(* LS Electric XG5000 project: POL(230517) *)
(* PLC NewPLC *)
(* module base 0 slot 0: FEnet:XGL-EFMT(B) (Fast Ethernet 통신 모듈, 전기 Master) *)
(* module base 1 slot 0: 아날로그입력 모듈:XGF-AC8A (A/D 전류 입력형 8채널) *)
(* module base 1 slot 1: 입력 모듈:XGI-D28A/B (DC 24V 입력, 64점 (전류소스 싱크공용/ 전류소스 입력)) *)
(* module base 1 slot 2: 입력 모듈:XGI-D28A/B (DC 24V 입력, 64점 (전류소스 싱크공용/ 전류소스 입력)) *)
(* module base 1 slot 3: 입력 모듈:XGI-D28A/B (DC 24V 입력, 64점 (전류소스 싱크공용/ 전류소스 입력)) *)
(* module base 1 slot 4: 입력 모듈:XGI-D28A/B (DC 24V 입력, 64점 (전류소스 싱크공용/ 전류소스 입력)) *)
(* module base 1 slot 5: 입력 모듈:XGI-D28A/B (DC 24V 입력, 64점 (전류소스 싱크공용/ 전류소스 입력)) *)
(* module base 1 slot 6: 출력 모듈:XGQ-TR8A/B (트랜지스터 출력, 64점 (0.1A용, 싱크출력/소스출력)) *)
(* module base 1 slot 7: 출력 모듈:XGQ-TR8A/B (트랜지스터 출력, 64점 (0.1A용, 싱크출력/소스출력)) *)
(* module base 2 slot 0: 출력 모듈:XGQ-TR8A/B (트랜지스터 출력, 64점 (0.1A용, 싱크출력/소스출력)) *)
(* module base 2 slot 1: 출력 모듈:XGQ-TR8A/B (트랜지스터 출력, 64점 (0.1A용, 싱크출력/소스출력)) *)
(* module base 2 slot 2: 출력 모듈:XGQ-TR8A/B (트랜지스터 출력, 64점 (0.1A용, 싱크출력/소스출력)) *)
(* module base 2 slot 3: 입력 모듈:XGI-D28A/B (DC 24V 입력, 64점 (전류소스 싱크공용/ 전류소스 입력)) *)
(* module base 2 slot 4: 입력 모듈:XGI-D28A/B (DC 24V 입력, 64점 (전류소스 싱크공용/ 전류소스 입력)) *)
(* module base 2 slot 5: 입력 모듈:XGI-D28A/B (DC 24V 입력, 64점 (전류소스 싱크공용/ 전류소스 입력)) *)
(* module base 2 slot 6: 출력 모듈:XGQ-TR8A/B (트랜지스터 출력, 64점 (0.1A용, 싱크출력/소스출력)) *)
(* module base 2 slot 7: Cnet:XGL-C42A/B (Cnet 통신 모듈(RS-422/485, RS-422/485)) *)
(* module base 2 slot 8: 아날로그출력 모듈:XGF-DC4A (D/A 전류 출력형 4채널) *)
VAR_GLOBAL
    TK101H : DWORD;
    TK101HH : DWORD;
    TK101L : DWORD;
    TK101LL : DWORD;
    TK101VAL : DWORD;
    TK102H : DWORD;
    TK102HH : DWORD;
    TK102L : DWORD;
    TK102LL : DWORD;
    TK102VAL : DWORD;
    TK103H : DWORD;
    TK103HH : DWORD;
    TK103L : DWORD;
    TK103LL : DWORD;
    TK103VAL : DWORD;
    TK104H : DWORD;
    TK104HH : DWORD;
    TK104L : DWORD;
    TK104LL : DWORD;
    TK104VAL : DWORD;
    TK105H : DWORD;
    TK105HH : DWORD;
    TK105L : DWORD;
    TK105LL : DWORD;
    TK105VAL : DWORD;
    TK106H : DWORD;
    TK106HH : DWORD;
    TK106L : DWORD;
    TK106LL : DWORD;
    TK106VAL : DWORD;
    TK107H : DWORD;
    TK107HH : DWORD;
    TK107L : DWORD;
    TK107LL : DWORD;
    TK107VAL : DWORD;
    TK108H : DWORD;
    TK108HH : DWORD;
    TK108L : DWORD;
    TK108LL : DWORD;
    TK108VAL : DWORD;
    TK109H : DWORD;
    TK109HH : DWORD;
    TK109L : DWORD;
    TK109LL : DWORD;
    TK109VAL : DWORD;
    TK110H : DWORD;
    TK110HH : DWORD;
    TK110L : DWORD;
    TK110LL : DWORD;
    TK110VAL : DWORD;
    TK111H : DWORD;
    TK111HH : DWORD;
    TK111L : DWORD;
    TK111LL : DWORD;
    TK111VAL : DWORD;
    TK112H : DWORD;
    TK112HH : DWORD;
    TK112L : DWORD;
    TK112LL : DWORD;
    TK112VAL : DWORD;
    TK113H : DWORD;
    TK113HH : DWORD;
    TK113L : DWORD;
    TK113LL : DWORD;
    TK113VAL : DWORD;
    _0000_ADDR_LNM AT %LW3761 : WORD; (* FEnet: LNM 정보(Ver 6.0이상) *)
    _0000_LINE_TOPOLOGY AT %LX60148 : BOOL; (* FEnet: Line topology 상태(Ver 6.0이상) *)
    _0100_CH0_ACT AT %UX1.0.16 : BOOL; (* 아날로그입력 모듈: 채널0 운전중 *)
    _0100_CH0_DATA AT %UW1.0.2 : INT; (* 아날로그입력 모듈: 채널0 변환값 *)
    _0100_CH0_IDD AT %UX1.0.160 : BOOL; (* 아날로그입력 모듈: 채널0 입력단선검출 *)
    _0100_CH1_ACT AT %UX1.0.17 : BOOL; (* 아날로그입력 모듈: 채널1 운전중 *)
    _0100_CH1_DATA AT %UW1.0.3 : INT; (* 아날로그입력 모듈: 채널1 변환값 *)
    _0100_CH1_IDD AT %UX1.0.161 : BOOL; (* 아날로그입력 모듈: 채널1 입력단선검출 *)
    _0100_CH2_ACT AT %UX1.0.18 : BOOL; (* 아날로그입력 모듈: 채널2 운전중 *)
    _0100_CH2_DATA AT %UW1.0.4 : INT; (* 아날로그입력 모듈: 채널2 변환값 *)
    _0100_CH2_IDD AT %UX1.0.162 : BOOL; (* 아날로그입력 모듈: 채널2 입력단선검출 *)
    _0100_CH3_ACT AT %UX1.0.19 : BOOL; (* 아날로그입력 모듈: 채널3 운전중 *)
    _0100_CH3_DATA AT %UW1.0.5 : INT; (* 아날로그입력 모듈: 채널3 변환값 *)
    _0100_CH3_IDD AT %UX1.0.163 : BOOL; (* 아날로그입력 모듈: 채널3 입력단선검출 *)
    _0100_CH4_ACT AT %UX1.0.20 : BOOL; (* 아날로그입력 모듈: 채널4 운전중 *)
    _0100_CH4_DATA AT %UW1.0.6 : INT; (* 아날로그입력 모듈: 채널4 변환값 *)
    _0100_CH4_IDD AT %UX1.0.164 : BOOL; (* 아날로그입력 모듈: 채널4 입력단선검출 *)
    _0100_CH5_ACT AT %UX1.0.21 : BOOL; (* 아날로그입력 모듈: 채널5 운전중 *)
    _0100_CH5_DATA AT %UW1.0.7 : INT; (* 아날로그입력 모듈: 채널5 변환값 *)
    _0100_CH5_IDD AT %UX1.0.165 : BOOL; (* 아날로그입력 모듈: 채널5 입력단선검출 *)
    _0100_CH6_ACT AT %UX1.0.22 : BOOL; (* 아날로그입력 모듈: 채널6 운전중 *)
    _0100_CH6_DATA AT %UW1.0.8 : INT; (* 아날로그입력 모듈: 채널6 변환값 *)
    _0100_CH6_IDD AT %UX1.0.166 : BOOL; (* 아날로그입력 모듈: 채널6 입력단선검출 *)
    _0100_CH7_ACT AT %UX1.0.23 : BOOL; (* 아날로그입력 모듈: 채널7 운전중 *)
    _0100_CH7_DATA AT %UW1.0.9 : INT; (* 아날로그입력 모듈: 채널7 변환값 *)
    _0100_CH7_IDD AT %UX1.0.167 : BOOL; (* 아날로그입력 모듈: 채널7 입력단선검출 *)
    _0208_CH0_ACT AT %UX2.8.16 : BOOL; (* 아날로그출력 모듈: 채널0 운전중 *)
    _0208_CH0_DATA AT %UW2.8.3 : INT; (* 아날로그출력 모듈: 채널0 입력값 *)
    _0208_CH0_ERR AT %UX2.8.0 : BOOL; (* 아날로그출력 모듈: 채널0 에러 *)
    _0208_CH0_OUTEN AT %UX2.8.32 : BOOL; (* 아날로그출력 모듈: 채널0 출력상태설정 *)
    _Auto_re_count : BOOL;
END_VAR

(* Comments on direct variables
%IX1.1.0	Power 0n_PB
%IX1.1.1	Power Off_PB
%IX1.1.2	Scada 선택 SL
%IX1.1.3	Panel 선택 SL
%IX1.1.5	Manual On_PB
%IX1.1.6	Auto On_PB
%IX1.1.7	Lamp Test PB
%IX1.1.8	Auto Stop (PANEL)
%IX1.1.9	Horn Reset PB
%IX1.1.10	In-TLV21601
%IX1.1.11	In-TLV21602
%IX1.1.12	In-TLV21701
%IX1.1.13	In-TLV21702
%IX1.1.14	In-TLV21801
%IX1.1.15	BCVF Open
%IX1.1.17	EM-Stop RESET
(PANEL)
%IX1.1.18	TK1-EM
%IX1.1.19	TK2-EM
%IX1.1.20	TK3-EM
%IX1.1.21	TK4-EM
%IX1.1.22	TK5-EM
%IX1.1.23	TK6-EM
%IX1.1.24	TK7-EM
%IX1.1.25	TK8-EM
%IX1.1.26	TK9-EM
%IX1.1.27	TK10-EM
%IX1.1.28	PUMP실-EM
%IX1.1.31	MAIN PANEL-EM PB
%IX1.1.32	TK-101 HLV  선택 PB
%IX1.1.33	VENT1 Trouble 
%IX1.1.34	VENT1 TURN 
%IX1.1.35	P101A OCR
%IX1.1.36	P101A Local Ready
%IX1.1.37	P101A Stop PB
%IX1.1.38	P101A Run PB
%IX1.1.39	P101B OCR
%IX1.1.40	P101B Local Ready
%IX1.1.41	P101B Stop_PB
%IX1.1.42	P101B Run_PB
%IX1.1.43	P101C OCR
%IX1.1.44	P101C Local Ready
%IX1.1.45	P101C Stop_PB
%IX1.1.46	P101C Run_PB
%IX1.1.47	TK-101 Clearance
%IX1.1.48	TK-102 HLV  선택 PB
%IX1.1.49	Vent2 Trouble
%IX1.1.50	Vent2 On
%IX1.1.51	P102A OCR
%IX1.1.52	P102A Local Ready
%IX1.1.53	P102A Stop_PB
%IX1.1.54	P102A Run_PB
%IX1.1.55	P102B OCR
%IX1.1.56	P102B Local Ready
%IX1.1.57	P102B Stop_PB
%IX1.1.58	P102B Run_PB
%IX1.1.59	P102C OCR
%IX1.1.60	P102C Local Ready
%IX1.1.61	P102C Stop_PB
%IX1.1.62	P102C Run_PB
%IX1.1.63	TK-102 Clearance
%IX1.2.0	TK-103 HLV 선택 PB
%IX1.2.1	Vent3 Trouble_in
%IX1.2.2	Vent3 On_in
%IX1.2.3	P103A OCR
%IX1.2.4	P103A Local Ready
%IX1.2.5	P103A Stop_PB
%IX1.2.6	P103A Run_PB
%IX1.2.7	P103B OCR
%IX1.2.8	P103B Local Ready
%IX1.2.9	P103B Stop_PB
%IX1.2.10	P103B Run_PB
%IX1.2.11	P103C OCR
%IX1.2.12	P103C Local Ready
%IX1.2.13	P103C Stop_PB
%IX1.2.14	P103C Run_PB
%IX1.2.15	TK-103 Clearance
%IX1.2.16	TK-104 HLV 선택 PB
%IX1.2.17	Vent4 Trouble_in
%IX1.2.18	Vent4 On_in
%IX1.2.19	P104A OCR
%IX1.2.20	P104A Local Ready
%IX1.2.21	P104A Stop_PB
%IX1.2.22	P104A Run_PB
%IX1.2.23	P104B OCR
%IX1.2.24	P104B Local Ready
%IX1.2.25	P104B Stop_PB
%IX1.2.26	P104B Run_PB
%IX1.2.27	P104C OCR
%IX1.2.28	P104C Local Ready
%IX1.2.29	P104C Stop_PB
%IX1.2.30	P104C Run_PB
%IX1.2.31	TK-104 Clearance
%IX1.2.32	TK-105 선택 [Panel]
%IX1.2.33	Vent5 Trouble_in
%IX1.2.34	Vent5 On_in
%IX1.2.35	P105A OCR
%IX1.2.36	P105A Local Ready
%IX1.2.37	P105A Stop_PB
%IX1.2.38	P105A Run_PB
%IX1.2.39	P105B OCR
%IX1.2.40	P105B Local Ready
%IX1.2.41	P105B Stop_PB
%IX1.2.42	P105B Run_PB
%IX1.2.43	P105C OCR
%IX1.2.44	P105C Local Ready
%IX1.2.45	P105C Stop_PB
%IX1.2.46	P105C Run_PB
%IX1.2.47	TK-105 Clearance
%IX1.2.48	TK-106 선택 [Panel]
%IX1.2.49	Vent6 Trouble_in
%IX1.2.50	Vent6 On_in
%IX1.2.51	P106A OCR
%IX1.2.52	P106A Local Ready
%IX1.2.53	P106A Stop_PB
%IX1.2.54	P106A Run_PB
%IX1.2.55	P106B OCR
%IX1.2.56	P106B Local Ready
%IX1.2.57	P106B Stop_PB
%IX1.2.58	P106B Run_PB
%IX1.2.59	P106C OCR
%IX1.2.60	P106C Local Ready
%IX1.2.61	P106C Stop_PB
%IX1.2.62	P106C Run_PB
%IX1.2.63	TK-106 Clearance
%IX1.3.0	TK-107 HLV 선택PB
%IX1.3.1	Vent7 Trouble
%IX1.3.2	Vent7 On
%IX1.3.3	P107A_OCR
%IX1.3.4	P107A_Local Ready
%IX1.3.5	P107A Stop_PB
%IX1.3.6	P107A Run_PB
%IX1.3.7	P107B_OCR
%IX1.3.8	P107B Local Ready
%IX1.3.9	P107B Stop_PB
%IX1.3.10	P107B Run_PB
%IX1.3.11	P107C_OCR
%IX1.3.12	P107C Local Ready
%IX1.3.13	P107C Stop_PB
%IX1.3.14	P107C Run_PB
%IX1.3.15	TK-107 Clearance
%IX1.3.16	TK-108 HLV 선택PB
%IX1.3.17	Vent8 Trouble_in
%IX1.3.18	Vent8 On_in
%IX1.3.19	P108A_OCR
%IX1.3.20	P108A_Local Ready
%IX1.3.21	P108A Stop_PB
%IX1.3.22	P108A Run_PB
%IX1.3.23	P108B_OCR
%IX1.3.24	P108B Local Ready
%IX1.3.25	P108B Stop_PB
%IX1.3.26	P108B Run_PB
%IX1.3.27	P108C_OCR
%IX1.3.28	P108C Local Ready
%IX1.3.29	P108C Stop_PB
%IX1.3.30	P108C Run_PB
%IX1.3.31	TK-108 Clearance
%IX1.3.32	TK-109 선택 [Panel]
%IX1.3.33	Vent9 Trouble_in
%IX1.3.34	Vent9 On_in
%IX1.3.35	P109A OCR
%IX1.3.36	P109A Local Ready
%IX1.3.37	P109A Stop_PB
%IX1.3.38	P109A Run_PB
%IX1.3.39	P109B OCR
%IX1.3.40	P109B Local Ready
%IX1.3.41	P109B Stop_PB
%IX1.3.42	P109B Run_PB
%IX1.3.43	P109C OCR
%IX1.3.44	P109C Local Ready
%IX1.3.45	P109C Stop_PB
%IX1.3.46	P109C Run_PB
%IX1.3.47	TK-109 Clearance
%IX1.3.48	TK-110 선택 [Panel]
%IX1.3.49	Vent10 Trouble_in
%IX1.3.50	Vent10 On_in
%IX1.3.51	P110A OCR
%IX1.3.52	P110A Local Ready
%IX1.3.53	P110A Stop_PB
%IX1.3.54	P110A Run_PB
%IX1.3.55	P110B OCR
%IX1.3.56	P110B Local Ready
%IX1.3.57	P110B Stop_PB
%IX1.3.58	P110B Run_PB
%IX1.3.59	P110C OCR
%IX1.3.60	P110C Local Ready
%IX1.3.61	P110C Stop_PB
%IX1.3.62	P110C Run_PB
%IX1.3.63	TK-110 Clearance
%IX1.4.0	HLVD-21301 FULL
%IX1.4.1	Water21301_in
%IX1.4.2	P111 OCR
%IX1.4.3	P111 Local S/W ON
%IX1.4.4	P111 Stop_PB
%IX1.4.5	P111 Run_PB
%IX1.4.6	Drain-111
Clearance
%IX1.4.7	HLVD-21401 FULL
%IX1.4.8	Water21401_in
%IX1.4.9	P112OCR
%IX1.4.10	P112 Local Ready
%IX1.4.11	P112 Stop_PB
%IX1.4.12	P112 Run_PB
%IX1.4.13	Drain-112
Clearance
%IX1.4.14	HLVD-21501 FULL
%IX1.4.15	Water21501_in
%IX1.4.16	P113 OCR
%IX1.4.17	P113 Local Ready
%IX1.4.18	Drain-113
Clearance
%IX1.4.19	UP201A OCR
%IX1.4.20	UP201A  Local Ready
%IX1.4.21	UP201A Stop_PB
%IX1.4.22	UP201A Run_PB
(PANEL)
%IX1.4.23	UP201B OCR
%IX1.4.24	UP201B Local Ready
%IX1.4.25	UP201B Stop_PB
%IX1.4.26	UP201B Run_PB
%IX1.4.27	UP202A OCR
%IX1.4.28	UP202A Local Ready
%IX1.4.29	UP202A Stop_PB
(PANEL)
%IX1.4.30	UP202A Run_PB
(PANEL)
%IX1.4.31	UP202B OCR
%IX1.4.32	UP202B Local Ready
%IX1.4.33	UP202B Stop_PB
%IX1.4.34	UP202B Run_PB
%IX1.4.35	UP203A OCR
%IX1.4.36	UP203A Local Ready
%IX1.4.37	UP203A Stop_PB
(PANEL)
%IX1.4.38	UP203A Run_PB
(PANEL)
%IX1.4.39	UP203B OCR
%IX1.4.40	UP203B Local Ready
%IX1.4.41	UP203B Stop_PB
%IX1.4.42	UP203B Run_PB
%IX1.4.45	PIPE LINE MOV20105 Close-PB
%IX1.4.47	PIPE LINE MOV 20105 Open-PB
%IX1.4.49	MOV20102 Over Torque
%IX1.4.50	MOV20102 Local
%IX1.4.51	MOV20102 Close-PB
%IX1.4.52	MOV20102 Close position
%IX1.4.53	MOV20102 Open-PB
%IX1.4.54	MOV20102 Open position
%IX1.4.55	MOV20103  Over Torque
%IX1.4.56	MOV20103  Local
%IX1.4.57	MOV20103 Close-PB
%IX1.4.58	MOV20103 Close position
%IX1.4.59	MOV20103 Open-PB
%IX1.4.60	MOV20103 Open position
%IX1.4.61	MOV20104 Over Torque
%IX1.4.62	MOV20104 Local
%IX1.4.63	MOV20104 Close-PB
%IX1.5.0	MOV20104 Close position
%IX1.5.1	MOV20104 Open-PB
%IX1.5.2	MOV20104 Open position
%IX1.5.3	MOV20105 Over Torque
%IX1.5.4	MOV20105 Local
%IX1.5.5	MOV20105 Close-PB
%IX1.5.6	MOV20105 Close position
%IX1.5.7	MOV20105 Open-PB
%IX1.5.8	MOV20105 Open position
%IX1.5.9	P101A Auto 1차 운전 선택 Switch(PANEL)
%IX1.5.10	P101B Auto 1차 운전 선택 Switch(PANEL)
%IX1.5.11	P102A Auto 1차 운전 선택 Switch(PANEL)
%IX1.5.12	P102B Auto 1차 운전 선택 Switch(PANEL)
%IX1.5.13	P103A Auto 1차 운전 선택 Switch(PANEL)
%IX1.5.14	P103B Auto 1차 운전 선택 Switch(PANEL)
%IX1.5.15	P104A Auto 1차 운전 선택 Switch(PANEL)
%IX1.5.16	P104B Auto 1차 운전 선택 Switch(PANEL)
%IX1.5.17	P107A Auto 1차 운전 선택 Switch(PANEL)
%IX1.5.18	P107B Auto 1차 운전 선택 Switch(PANEL)
%IX1.5.19	P108A Auto 1차 운전 선택 Switch(PANEL)
%IX1.5.20	P108B Auto 1차 운전 선택 Switch(PANEL)
%IX1.5.25	P101A Auto 2차 운전 선택 Switch(PANEL)
%IX1.5.26	P101B Auto 2차 운전 선택 Switch(PANEL)
%IX1.5.27	P102A Auto 2차 운전 선택 Switch(PANEL)
%IX1.5.28	P102B Auto 2차 운전 선택 Switch(PANEL)
%IX1.5.29	P103A Auto 2차 운전 선택 Switch(PANEL)
%IX1.5.30	P103B Auto 2차 운전 선택 Switch(PANEL)
%IX1.5.31	P104A Auto 2차 운전 선택 Switch(PANEL)
%IX1.5.32	P104B Auto 2차 운전 선택 Switch(PANEL)
%IX1.5.33	P107A Auto 2차 운전 선택 Switch(PANEL)
%IX1.5.34	P107B Auto 2차 운전 선택 Switch(PANEL)
%IX1.5.35	P108A Auto 2차 운전 선택 Switch(PANEL)
%IX1.5.36	P108B Auto 2차 운전 선택 Switch(PANEL)
%IX1.5.41	P113 Stop_PB
%IX1.5.42	P113 Run_PB
%IX1.5.43	Auto Start PB
%IX1.5.48	RTU#1 
OPEN SIG
TO HS_PLC
%IX1.5.49	RTU#2
OPEN SIG
TO HS_PLC
%IX1.5.50	RTU#3
OPEN SIG
TO HS_PLC
%IX1.5.51	RTU#4
OPEN SIG
TO HS_PLC
%IX1.5.52	RTU#5
OPEN SIG
TO HS_PLC
%IX1.5.53	PRV OPEN SIG TO HS_PLC
%IX2.3.0	P101A Flow Switch
%IX2.3.1	P101A THERMOSTAT
%IX2.3.2	P101B Flow Switch
%IX2.3.3	P101B THERMOSTAT
%IX2.3.4	P101C Flow Switch
%IX2.3.5	P101C Thermostat
%IX2.3.6	P102A Flow Switch
%IX2.3.7	P102A Thermostat
%IX2.3.8	P102B Flow Switch
%IX2.3.9	P102B Thermostat
%IX2.3.10	P102C Flow Switch
%IX2.3.11	P102C Thermostat
%IX2.3.12	P103A Flow Switch
%IX2.3.13	P103A Thermostat
%IX2.3.14	P103B Flow Switch
%IX2.3.15	P103B Thermostat
%IX2.3.16	P103C Flow Switch
%IX2.3.17	P103C Thermostat
%IX2.3.18	P104A Flow Switch
%IX2.3.19	P104A Thermostat
%IX2.3.20	P104B Flow Switch
%IX2.3.21	P104B Thermostat
%IX2.3.22	P104C Flow Switch
%IX2.3.23	P104C Thermostat
%IX2.3.24	UP201A Flow Switch
%IX2.3.25	UP201A Thermostat
%IX2.3.26	UP201B Flow Switch
%IX2.3.27	UP201B Thermostat
%IX2.3.28	P105A Flow Switch
%IX2.3.29	P105A Thermostat
%IX2.3.30	P105B Flow Switch
%IX2.3.31	P105B Thermostat
%IX2.3.32	P105C Flow Switch
%IX2.3.33	P105C Thermostat
%IX2.3.34	P106A Flow Switch
%IX2.3.35	P106A Thermostat
%IX2.3.36	P106B Flow Switch
%IX2.3.37	P106B Thermostat
%IX2.3.38	P106C Flow Switch
%IX2.3.39	P106C Thermostat
%IX2.3.40	P107A Flow Switch Alarm
%IX2.3.41	P107A Thermostat
%IX2.3.42	P107B Flow Switch Alarm
%IX2.3.43	P107B Thermostat
%IX2.3.44	P107C Flow Switch Alarm
%IX2.3.45	P107C Thermostat
%IX2.3.46	P108A Flow Switch Alarm
%IX2.3.47	P108A Thermostat
%IX2.3.48	P108B Flow Switch Alarm
%IX2.3.49	P108B Thermostat
%IX2.3.50	P108C Flow Switch Alarm
%IX2.3.51	P108C Thermostat
%IX2.3.52	P109A Flow Switch
%IX2.3.53	P109A Thermostat
%IX2.3.54	P109B Flow Switch
%IX2.3.55	P109B Thermostat
%IX2.3.56	P109C Flow Switch
%IX2.3.57	P109C Thermostat
%IX2.3.58	P110A Flow Switch
%IX2.3.59	P110A Thermostat
%IX2.3.60	P110B Flow Switch
%IX2.3.61	P110B Thermostat
%IX2.3.62	P110C Flow Switch
%IX2.3.63	P110C Thermostat
%IX2.4.0	P111 Flow Switch
%IX2.4.1	TK-111 Thermostat
%IX2.4.2	P112 Flow Switch
%IX2.4.3	TK-112 Thermostat
%IX2.4.4	P113 Flow Switch
%IX2.4.5	TK-113 Thermostat
%IX2.4.6	UP202A Flow Switch
%IX2.4.7	UP202A Thermostat
%IX2.4.8	UP202B Flow Switch
%IX2.4.9	UP202B Thermostat
%IX2.4.10	UP203A Flow Switch
%IX2.4.11	UP203A Thermostat
%IX2.4.12	UP203B Flow Switch
%IX2.4.13	UP203B Thermostat
%IX2.4.14	TK-101A PUMP ON MCC MC ON SIG
%IX2.4.15	TK-101B PUMP ON MCC MC ON SIG
%IX2.4.16	TK-101C PUMP ON MCC MC ON SIG
%IX2.4.17	TK-102A PUMP ON MCC MC ON SIG
%IX2.4.18	TK-102B PUMP ON MCC MC ON SIG
%IX2.4.19	TK-102C PUMP ON MCC MC ON SIG
%IX2.4.20	TK-103A PUMP ON MCC MC ON SIG
%IX2.4.21	TK-103B PUMP ON MCC MC ON SIG
%IX2.4.22	TK-103C PUMP ON MCC MC ON SIG
%IX2.4.23	TK-104A PUMP ON MCC MC ON SIG
%IX2.4.24	TK-104B PUMP ON MCC MC ON SIG
%IX2.4.25	TK-104C PUMP ON MCC MC ON SIG
%IX2.4.26	TK-105A PUMP ON MCC MC ON SIG
%IX2.4.27	TK-105B PUMP ON MCC MC ON SIG
%IX2.4.28	TK-105C PUMP ON MCC MC ON SIG
%IX2.4.29	TK-106A PUMP ON MCC MC ON SIG
%IX2.4.30	TK-106B PUMP ON MCC MC ON SIG
%IX2.4.31	TK-106C PUMP ON MCC MC ON SIG
%IX2.4.32	TK-107A PUMP ON MCC MC ON SIG
%IX2.4.33	TK-107B PUMP ON MCC MC ON SIG
%IX2.4.34	TK-107C PUMP ON MCC MC ON SIG
%IX2.4.35	TK-108A PUMP ON MCC MC ON SIG
%IX2.4.36	TK-108B PUMP ON MCC MC ON SIG
%IX2.4.37	TK-108C PUMP ON MCC MC ON SIG
%IX2.4.38	TK-109A PUMP ON MCC MC ON SIG
%IX2.4.39	TK-109B PUMP ON MCC MC ON SIG
%IX2.4.40	TK-109C PUMP ON MCC MC ON SIG
%IX2.4.41	TK-110A PUMP ON MCC MC ON SIG
%IX2.4.42	TK-110B PUMP ON MCC MC ON SIG
%IX2.4.43	TK-110C PUMP ON MCC MC ON SIG
%IX2.4.44	DRAIN TK-111 PUMP ON MCC MC ON SIG
%IX2.4.45	DRAIN TK-112 PUMP ON MCC MC ON SIG
%IX2.4.46	DRAIN TK-113 PUMP ON MCC MC ON SIG
%IX2.4.47	UP201A PUMP ON MCC MC ON SIG
%IX2.4.48	UP201B PUMP ON MCC MC ON SIG
%IX2.4.49	UP202A PUMP ON MCC MC ON SIG
%IX2.4.50	UP202B PUMP ON MCC MC ON SIG
%IX2.4.51	UP203A PUMP ON MCC MC ON SIG
%IX2.4.52	UP203B PUMP ON MCC MC ON SIG
%IX2.4.53	UP201A  Local Ready   (PANTO_1)
%IX2.4.54	UP201A RUN_PB
(PANTO_1)
%IX2.4.55	UP201A STOP_PB
(PANTO_1)
%IX2.4.56	PANTO1_EM
%IX2.4.57	UP201B  Local Ready   (PANTO_2)
%IX2.4.58	UP201B RUN_PB
(PANTO_2)
%IX2.4.59	UP201B STOP_PB
(PANTO_2)
%IX2.4.60	PANTO2_EM
%IX2.4.61	UP202A  Local Ready   (PANTO_3)
%IX2.4.62	UP202A RUN_PB
(PANTO_3)
%IX2.4.63	UP202A STOP_PB
(PANTO_3)
%IX2.5.0	PANTO3_EM
%IX2.5.1	UP203A  Local Ready   (PANTO_4)
%IX2.5.2	UP203A RUN_PB
(PANTO_4)
%IX2.5.3	UP203A STOP_PB
(PANTO_4)
%IX2.5.4	PANTO4_EM
%IX2.5.5	UP203B  Local Ready   (PANTO_5)
%IX2.5.6	UP203B RUN_PB
(PANTO_5)
%IX2.5.7	UP203B STOP_PB
(PANTO_5)
%IX2.5.8	PANTO5_EM
%IX2.5.9	Drain TK-111 Pressure SW
%IX2.5.10	Drain TK-112 Pressure SW
%IX2.5.11	Drain TK-113 Pressure SW
%IX2.5.12	LDS ALARM
%IX2.5.13	LDS PNL EM
%IX2.5.14	TK-108 LEAK - 1 ON
%IX2.5.15	TK-108 LEAK - 2 ON
%IX2.5.16	TK-108 LEAK - 3 ON
%IX2.5.17	TK-108 LEAK - 4 ON
%QX1.6.0	Power On Lamp
%QX1.6.1	Power Off Lamp
%QX1.6.2	SCADA 선택 Lamp
%QX1.6.3	Panel 선택 Lamp
%QX1.6.4	BUZZER Stop Lamp
%QX1.6.5	Manual 선택 Lamp
%QX1.6.6	Auto 선택 Lamp
%QX1.6.7	Auto Stop Lamp
%QX1.6.8	외부 HORN
%QX1.6.9	BPCV
%QX1.6.10	CVP
%QX1.6.11	EV_SOL
%QX1.6.12	CVP Lamp
%QX1.6.13	EV Lamp
%QX1.6.14	In-TLV21601 Lamp
%QX1.6.15	In-TLV21602 Lamp
%QX1.6.16	In-TLV21701 Lamp
%QX1.6.17	In-TLV21702 Lamp
%QX1.6.18	In-TLV21801Lamp
%QX1.6.19	BCVF 20101 Lamp
%QX1.6.20	BPCV Lamp
%QX1.6.21	TK103-EM Lamp
%QX1.6.22	TK104-EM Lamp
%QX1.6.23	TK105-EM Lamp
%QX1.6.24	TK106-EM Lamp
%QX1.6.25	TK107-EM Lamp
%QX1.6.26	TK108-EM Lamp
%QX1.6.27	TK109-EM Lamp
%QX1.6.28	TK110-EM Lamp
%QX1.6.29	TK101-EM Lamp
%QX1.6.30	TK102-EM Lamp
%QX1.6.31	EM-Stop RESET Lamp
%QX1.6.32	MAIN PANEL EM Lamp
%QX1.6.33	Lamp Test Lamp
%QX1.6.34	Auto Start Lamp
%QX1.6.38	PIT_01A
TROUBLE
[회수압력]
%QX1.6.39	PIT_01B
TROUBLE
[수령압력]
%QX1.6.40	PIT_02A
TROUBLE
[불출압력]
%QX1.6.41	PIT_02B
TROUBLE
[불출압력]
%QX1.6.42	FIT_01A
TROUBLE
[불출유량]
%QX1.6.43	FIT_01B
TROUBLE
[불출유량]
%QX1.6.44	FIT_03A
TROUBLE
[회수유량]
%QX1.6.45	FIT_03B
TROUBLE
[회수유량]
%QX1.6.46	A-SIDE PLC RUN Lamp
%QX1.6.47	B-SIDE PLC RUN Lamp
%QX1.6.48	HLV20301 TK101 Open
%QX1.6.49	VENT1 Trouble Lamp
%QX1.6.50	VENT1 TURN Lamp
%QX1.6.51	P101A Trouble Lamp
%QX1.6.52	P101A Local Lamp
%QX1.6.53	P101A Stop Lamp
%QX1.6.54	P101A Run
%QX1.6.55	P101B Trouble Lamp
%QX1.6.56	P101B Local Lamp
%QX1.6.57	P101B Stop Lamp
%QX1.6.58	P101B Run
%QX1.6.59	P101C Trouble Lamp
%QX1.6.60	P101C Local Lamp
%QX1.6.61	P101C Stop Lamp
%QX1.6.62	P101C Run
%QX1.6.63	HLV20401 TK102 Open
%QX1.7.0	Vent2 Trouble Lamp
%QX1.7.1	TK102 Ventilator Lamp
%QX1.7.2	P102A Trouble Lamp
%QX1.7.3	P102A Local Lamp
%QX1.7.4	P102A Stop Lamp
%QX1.7.5	P102A Run
%QX1.7.6	P102B Trouble Lamp
%QX1.7.7	P102B Local Lamp
%QX1.7.8	P102B Stop Lamp
%QX1.7.9	P102B Run
%QX1.7.10	P102C Trouble Lamp
%QX1.7.11	P102C Local Lamp
%QX1.7.12	P102C Stop Lamp
%QX1.7.13	P102C Run
%QX1.7.14	HLV20501 TK103 Open
%QX1.7.15	Vent3 Trouble Lamp
%QX1.7.16	TK103 Ventilator Lamp
%QX1.7.17	P103A Trouble Lamp
%QX1.7.18	P103A Local Lamp
%QX1.7.19	P103A Stop Lamp
%QX1.7.20	P103A Run
%QX1.7.21	P103B Trouble Lamp
%QX1.7.22	P103B Local Lamp
%QX1.7.23	P103B Stop Lamp
%QX1.7.24	P103B Run
%QX1.7.25	P103C Trouble Lamp
%QX1.7.26	P103C Local Lamp
%QX1.7.27	P103C Stop Lamp
%QX1.7.28	P103C Run
%QX1.7.29	HLV20601 TK104 Open
%QX1.7.30	Vent4 Trouble Lamp
%QX1.7.31	TK104 Ventilator Lamp
%QX1.7.32	P104A Trouble Lamp
%QX1.7.33	P104A Local Lamp
%QX1.7.34	P104A Stop Lamp
%QX1.7.35	P104A Run
%QX1.7.36	P104B Trouble Lamp
%QX1.7.37	P104B Local Lamp
%QX1.7.38	P104B Stop Lamp
%QX1.7.39	P104B Run
%QX1.7.40	P104C Trouble Lamp
%QX1.7.41	P104C Local Lamp
%QX1.7.42	P104C Stop Lamp
%QX1.7.43	P104C Run
%QX1.7.44	HLV20701 TK105 Open
%QX1.7.45	Vent5 Trouble Lamp
%QX1.7.46	TK105 Ventilator Lamp
%QX1.7.47	P105A Trouble Lamp
%QX1.7.48	P105A Local Lamp
%QX1.7.49	P105A Stop Lamp
%QX1.7.50	P105A Run 
%QX1.7.51	P105B Trouble Lamp
%QX1.7.52	P105B Local Lamp
%QX1.7.53	P105B Stop Lamp
%QX1.7.54	P105B Run
%QX1.7.55	P105C Trouble Lamp
%QX1.7.56	P105C Local Lamp
%QX1.7.57	P105C Stop Lamp
%QX1.7.58	P105C Run
%QX1.7.59	HLV20801 TK106 Open
%QX1.7.60	Vent6 Trouble Lamp
%QX1.7.61	TK106 Ventilator Lamp
%QX1.7.62	P106A Trouble Lamp
%QX1.7.63	P106A Local Lamp
%QX1.9.60	PIPE LINE MOV 20101 Trouble
%QX1.9.61	PIPE LINE MOV 20101 Local
%QX1.9.62	PIPE LINE MOV 20105 Close Lamp
%QX1.9.63	MOV20101 Close
%QX1.10.0	PIPE LINE MOV 20101 Open Lamp
%QX1.10.1	MOV20101 Open
%QX2.0.0	P106A Stop Lamp
%QX2.0.1	P106A Run
%QX2.0.2	P106B Trouble Lamp
%QX2.0.3	P106B Local Lamp
%QX2.0.4	P106B Stop Lamp
%QX2.0.5	P106B Run
%QX2.0.6	P106C Trouble Lamp
%QX2.0.7	P106C Local Lamp
%QX2.0.8	P106C Stop Lamp
%QX2.0.9	P106C Run
%QX2.0.10	HLV20901 TK107 Open
%QX2.0.11	Vent7 Trouble Lamp
%QX2.0.12	TK107 Ventilator Lamp
%QX2.0.13	P107A Trouble Lamp
%QX2.0.14	P107A Local Lamp
%QX2.0.15	P107A Stop
%QX2.0.16	P107A Run
%QX2.0.17	P107B Trouble Lamp
%QX2.0.18	P107B Local Lamp
%QX2.0.19	P107B Stop
%QX2.0.20	P107B Run
%QX2.0.21	P107C Trouble Lamp
%QX2.0.22	P107C Local Lamp
%QX2.0.23	P107C Stop
%QX2.0.24	P107C Run
%QX2.0.25	HLV21001 TK108 Open
%QX2.0.26	Vent8 Trouble Lamp
%QX2.0.27	TK108 Ventilator Lamp
%QX2.0.28	P108A Trouble Lamp
%QX2.0.29	P108A Local Lamp
%QX2.0.30	P108A Stop Lamp
%QX2.0.31	P108A Run
%QX2.0.32	P108B Trouble Lamp
%QX2.0.33	P108B Local Lamp
%QX2.0.34	P108B Stop Lamp
%QX2.0.35	P108B Run
%QX2.0.36	P108C Trouble Lamp
%QX2.0.37	P108C Local Lamp
%QX2.0.38	P108C Stop Lamp
%QX2.0.39	P108C Run
%QX2.0.40	HLV21101 TK109 Open
%QX2.0.41	Vent9 Trouble Lamp
%QX2.0.42	TK109 Ventilator
%QX2.0.43	P109A Trouble Lamp
%QX2.0.44	P109A Local Lamp
%QX2.0.45	P109A Stop Lamp
%QX2.0.46	P109A Run
%QX2.0.47	P109B Trouble Lamp
%QX2.0.48	P109B Local Lamp
%QX2.0.49	P109B Stop Lamp
%QX2.0.50	P109B Run
%QX2.0.51	P109C Trouble Lamp
%QX2.0.52	P109C Local Lamp
%QX2.0.53	P109C Stop Lamp
%QX2.0.54	P109C Run
%QX2.0.55	HLV21201 TK110 Open
%QX2.0.56	Vent10 Trouble Lamp
%QX2.0.57	TK110 Ventilator Lamp
%QX2.0.58	P110A Trouble Lamp
%QX2.0.59	P110A Local Lamp
%QX2.0.60	P110A Stop Lamp
%QX2.0.61	P110A Run
%QX2.0.62	P110B Trouble Lamp
%QX2.0.63	P110B Local Lamp
%QX2.1.0	P110B Stop Lamp
%QX2.1.1	P110B Run
%QX2.1.2	P110C Trouble Lamp
%QX2.1.3	P110C Local Lamp
%QX2.1.4	P110C Stop Lamp
%QX2.1.5	P110C Run
%QX2.1.6	HLVD FULL 21301 Lamp
%QX2.1.7	Water21301 Lamp
%QX2.1.8	P111 Trouble Lamp
%QX2.1.9	DRAIN TK-111 Local Lamp
%QX2.1.10	P111 Stop Lamp
%QX2.1.11	P111 Run
%QX2.1.12	DRAIN TANK111 Level 95%   HH Lamp
%QX2.1.13	DRAIN TANK111 Level 90%   H Lamp
%QX2.1.14	DRAIN TANK111 Level 정상 Lamp
%QX2.1.15	DRAIN TANK111 Level 15%   L  Lamp
%QX2.1.16	DRAIN TANK111 Level 10%   LL Lamp
%QX2.1.17	HLVD MAX 21401 Lamp
%QX2.1.18	Water21401 Lamp
%QX2.1.19	P112 Trouble Lamp
%QX2.1.20	DRAIN TK-112 Local Lamp
%QX2.1.21	P112 Stop Lamp
%QX2.1.22	P112 Run
%QX2.1.23	DRAIN TANK112 Level 95%   HH  Lamp
%QX2.1.24	DRAIN TANK112 Level 90%   H Lamp
%QX2.1.25	DRAIN TANK112 Level 정상 Lamp
%QX2.1.26	DRAIN TANK112 Level 15%   L Lamp
%QX2.1.27	DRAIN TANK112 Level 10%   LL  Lamp
%QX2.1.28	HLVD MAX 21501 Lamp
%QX2.1.29	Water21501 Lamp
%QX2.1.30	P113 Trouble Lamp
%QX2.1.31	DRAIN TANK113 Level 95%   HH Lamp
%QX2.1.32	DRAIN TANK113 Level 90%   H Lamp
%QX2.1.33	DRAIN TANK113 Level 정상 Lamp
%QX2.1.34	DRAIN TANK113 Level 15%   L Lamp
%QX2.1.35	DRAIN TANK113 Level 10%   LL Lamp
%QX2.1.36	UP201A Trouble Lamp
%QX2.1.37	UP201A Local Lamp
(Pump room)
%QX2.1.38	UP201A Stop Lamp
%QX2.1.39	UP201A Run
%QX2.1.40	UP201B Trouble Lamp
%QX2.1.41	UP201B Local Lamp
(Pump room)
%QX2.1.42	UP201B Stop Lamp
%QX2.1.43	UP201B Run
%QX2.1.44	UP202A Trouble Lamp
%QX2.1.45	UP202A Local Lamp
(Pump room)
%QX2.1.46	UP202A Stop Lamp
%QX2.1.47	UP202A Run
%QX2.1.48	UP202B Trouble Lamp
%QX2.1.49	UP202B Local Lamp
%QX2.1.50	UP202B Stop Lamp
%QX2.1.51	UP202B Run
%QX2.1.52	UP203A Trouble Lamp
%QX2.1.53	UP203A Local Lamp
(Pump room)
%QX2.1.54	UP203A Stop Lamp
%QX2.1.55	UP203A Run
%QX2.1.56	UP203B Trouble Lamp
%QX2.1.57	UP203B Local Lamp
(Pump room)
%QX2.1.58	UP203B Stop Lamp
%QX2.1.59	UP203B Run
%QX2.2.2	MOV20102 Trouble Lamp
%QX2.2.3	MOV20102 Local Lamp
%QX2.2.4	MOV20102 Close Lamp
%QX2.2.5	MOV20102 Close
%QX2.2.6	MOV20102 Open Lamp
%QX2.2.7	MOV20102 Open
%QX2.2.8	MOV20103 Trouble Lamp
%QX2.2.9	MOV20103 Local Lamp
%QX2.2.10	MOV20103 Close Lamp
%QX2.2.11	MOV20103 Close
%QX2.2.12	MOV20103 Open Lamp
%QX2.2.13	MOV20103 Open
%QX2.2.14	MOV20104 Trouble Lamp
%QX2.2.15	MOV20104 Local Lamp
%QX2.2.16	MOV20104 Close Lamp
%QX2.2.17	MOV20104 Close
%QX2.2.18	MOV20104 Open Lamp
%QX2.2.19	MOV20104 Open 
%QX2.2.20	MOV20105 Trouble Lamp
%QX2.2.21	MOV20105 Local Lamp
%QX2.2.22	MOV20105 Close Lamp
%QX2.2.23	MOV20105 Close 
%QX2.2.24	MOV20105 Open Lamp
%QX2.2.25	MOV20105 Open 
%QX2.2.26	P101A Auto 1차 운전 선택 Lamp
%QX2.2.27	P101B Auto 1차 운전 선택 Lamp
%QX2.2.28	P102A Auto 1차 운전 선택 Lamp
%QX2.2.29	P102B Auto 1차 운전 선택 Lamp
%QX2.2.30	P103A Auto 1차 운전 선택 Lamp
%QX2.2.31	P103B Auto 1차 운전 선택 Lamp
%QX2.2.32	P104A Auto 1차 운전 선택 Lamp
%QX2.2.33	P104B Auto 1차 운전 선택 Lamp
%QX2.2.34	P107A Auto 1차 운전 선택 Lamp
%QX2.2.35	P107B Auto 1차 운전 선택 Lamp
%QX2.2.36	P108A Auto 1차 운전 선택 Lamp
%QX2.2.37	P108B Auto 1차 운전 선택 Lamp
%QX2.2.42	P101A Auto 2차 운전 선택 Lamp
%QX2.2.43	P101B Auto 2차 운전 선택 Lamp
%QX2.2.44	P102A Auto 2차 운전 선택 Lamp
%QX2.2.45	P102B Auto 2차 운전 선택 Lamp
%QX2.2.46	P103A Auto 2차 운전 선택 Lamp
%QX2.2.47	P103B Auto 2차 운전 선택 Lamp
%QX2.2.48	P104A Auto 2차 운전 선택 Lamp
%QX2.2.49	P104B Auto 2차 운전 선택 Lamp
%QX2.2.50	P107A Auto 2차 운전 선택 Lamp
%QX2.2.51	P107B Auto 2차 운전 선택 Lamp
%QX2.2.52	P108A Auto 2차 운전 선택 Lamp
%QX2.2.53	P108B Auto 2차 운전 선택 Lamp
%QX2.2.58	DRAIN TK-113 Local Lamp
%QX2.2.59	P113 Stop Lamp
%QX2.2.60	P113 Run
%QX2.6.0	P101A Run Lamp
%QX2.6.1	P101B Run Lamp
%QX2.6.2	P101C Run Lamp
%QX2.6.3	P102A Run Lamp
%QX2.6.4	P102B Run Lamp
%QX2.6.5	P102C Run Lamp
%QX2.6.6	P103A Run Lamp
%QX2.6.7	P103B Run Lamp
%QX2.6.8	P103C Run Lamp
%QX2.6.9	P104A Run Lamp
%QX2.6.10	P104B Run Lamp
%QX2.6.11	P104C Run Lamp
%QX2.6.12	P105A Run Lamp
%QX2.6.13	P105B Run Lamp
%QX2.6.14	P105C Run Lamp
%QX2.6.15	P106A Run Lamp
%QX2.6.16	P106B Run Lamp
%QX2.6.17	P106C Run Lamp
%QX2.6.18	P107A Run Lamp
%QX2.6.19	P107B Run Lamp
%QX2.6.20	P107C Run Lamp
%QX2.6.21	P108A Run Lamp
%QX2.6.22	P108B Run Lamp
%QX2.6.23	P108C Run Lamp
%QX2.6.24	P109A Run Lamp
%QX2.6.25	P109B Run Lamp
%QX2.6.26	P109C Run Lamp
%QX2.6.27	P110A Run Lamp
%QX2.6.28	P110B Run Lamp
%QX2.6.29	P110C Run Lamp
%QX2.6.30	P111 Run Lamp
%QX2.6.31	P112 Run Lamp
%QX2.6.32	P113 Run Lamp
%QX2.6.33	UP201A Run Lamp
%QX2.6.34	UP201B Run Lamp
%QX2.6.35	UP202A Run Lamp
%QX2.6.36	UP202B Run Lamp
%QX2.6.37	UP203A Run Lamp
%QX2.6.38	UP203B Run Lamp
%QX2.6.39	HLV20301 TK101 Open Lamp
%QX2.6.40	HLV20301 TK102 Open Lamp
%QX2.6.41	HLV20501 TK103 Open Lamp
%QX2.6.42	HLV20601 TK104 Open Lamp
%QX2.6.43	HLV20701 TK105 Open Lamp
%QX2.6.44	HLV20801 TK106 Open Lamp
%QX2.6.45	HLV20901 TK107 Open Lamp
%QX2.6.46	HLV21001 TK108 Open Lamp
%QX2.6.47	HLV21101 TK109 Open Lamp
%QX2.6.48	HLV21201 TK110 Open Lamp
%QX2.6.49	PUMP실-EM Lamp
%QX2.6.50	P107A Stop Lamp
%QX2.6.51	P107B Stop Lamp
%QX2.6.52	P107C Stop Lamp
%QX2.6.53	내부 HORN
%QX2.6.54	TOTAL EM [MCC Power Off]
%MX0	A-SIDE PLC RUN to SCADA
%MX1	B-SIDE PLC RUN to SCADA
%MX2	ARES 수령중 HH & HLV OPEN
%MX3	POL NMR5000 통신이상 신호
%MX4	POL NMR 통신이상
%MX5	TK-101 수령 중
HH & HLV OPEN
%MX6	TK-102 수령 중
HH & HLV OPEN
%MX7	TK-103 수령 중
HH & HLV OPEN
%MX8	TK-104 수령 중
HH & HLV OPEN
%MX9	TK-107 수령 중
HH & HLV OPEN
%MX10	TK-110 수령 중
HH & HLV OPEN
%MX12	Auto Restart Alarm
%MX13	Power on [Scada]
%MX14	HLV_RESET [SCADA]
%MX15	120대대 TLV OPEN
%MX16	Bottom Tap manu
[수불출 현황 to SCADA]
%MX17	Bottom Tap manu
[jp-8,diesel to SCADA]
%MX64	Manual [SCADA]
%MX65	Auto [SCADA]
%MX66	Auto Start (SCADA)
%MX67	Auto Stop (SCADA)
%MX68	EM-Stop RESET
(SCADA)
%MX69	Horn Reset SCADA
%MX70	TK-101 선택 
(SCADA)
%MX71	TK-102 선택 
(SCADA)
%MX72	TK-103 선택 
(SCADA)
%MX73	TK-104 Auto 선택 
(SCADA)
%MX74	TK-107 Auto 선택 
(SCADA)
%MX75	TK-108 선택 
(SCADA)
%MX76	TK-105 선택 [SCADA]
%MX77	TK-106 선택 [SCADA]
%MX78	TK-109 선택 [SCADA]
%MX79	TK-110 선택 [SCADA]
%MX80	TK-107 선택 SCADA    (수령)
%MX81	TK-108 선택 SCADA   (수령)
%MX82	LDS ALARM
%MX100	CH0 단선검출
%MX101	CH1 단선검출
%MX102	CH2 단선검출
%MX103	CH3 단선검출
%MX104	CH4 단선검출
%MX105	CH5 단선검출
%MX106	CH6 단선검출
%MX107	CH7 단선검출
%MX110	ARES PUMP Running CHECK
%MX128	P101A Run SCADA
%MX129	P101A Stop SCADA
%MX132	P101B Run SCADA
%MX133	P101B Stop SCADA
%MX136	P101C Run SCADA
%MX137	P101C Stop SCADA
%MX140	P102A Run SCADA
%MX141	P102A Stop SCADA
%MX144	P102B Run SCADA
%MX145	P102B Stop SCADA
%MX148	P102C Run SCADA
%MX149	P102C Stop SCADA
%MX152	P103A Run SCADA
%MX153	P103A Stop SCADA
%MX156	P103B Run SCADA
%MX157	P103B Stop SCADA
%MX160	P103C Run SCADA
%MX161	P103C Stop SCADA
%MX164	P104A Run SCADA
%MX165	P104A Stop SCADA
%MX168	P104B Run SCADA
%MX169	P104B Stop SCADA
%MX172	P104C Run SCADA
%MX173	P104C Stop SCADA
%MX176	P105A Run SCADA
%MX177	P105A Stop SCADA
%MX180	P105B Run SCADA
%MX181	P105B Stop SCADA
%MX192	P105C Run SCADA
%MX193	P105C Stop SCADA
%MX196	P106A Run SCADA
%MX197	P106A Stop SCADA
%MX202	P106B Run SCADA
%MX203	P106B Stop SCADA
%MX206	P106C Run SCADA
%MX207	P106C Stop SCADA
%MX210	P107A Run SCADA
%MX211	P107A Stop SCADA
%MX214	P107B Run SCADA
%MX215	P107B Stop SCADA
%MX218	P107C Run SCADA
%MX219	P107C Stop SCADA
%MX222	P108A Run SCADA
%MX223	P108A Stop SCADA
%MX226	P108B Run SCADA
%MX227	P108B Stop SCADA
%MX230	P108C Run SCADA
%MX231	P108C Stop SCADA
%MX234	P109A Run SCADA
%MX235	P109A Stop SCADA
%MX238	P109B Run SCADA
%MX239	P109B Stop SCADA
%MX242	P109C Run SCADA
%MX243	P109C Stop SCADA
%MX246	P110A Run SCADA
%MX247	P110A Stop SCADA
%MX250	P110B Run SCADA
%MX251	P110B Stop SCADA
%MX254	P110C Run SCADA
%MX255	P110C Stop SCADA
%MX256	DRAIN TK-111 Run SCADA
%MX257	DRAIN TK-111 Stop SCADA
%MX260	DRAIN TK-112 Run SCADA
%MX261	DRAIN TK-112 Stop SCADA
%MX264	DRAIN TK-113 Run SCADA
%MX265	DRAIN TK-113 Stop SCADA
%MX266	MOV 20103     Open  (SCADA)
%MX267	MOV 20103    Close  (SCADA)
%MX270	MOV 20104     Open  (SCADA)
%MX271	MOV 20104    Close  (SCADA)
%MX274	MOV 20102     Open  (SCADA)
%MX275	MOV 20102    Close  (SCADA)
%MX278	MOV 20105     Open  (SCADA)
%MX279	MOV 20105    Close  (SCADA)
%MX282	MOV 20101     Open  (SCADA)
%MX283	MOV 20101    Close  (SCADA)
%MX286	UP201A    Run  (SCADA)
%MX287	UP201A   Stop  (SCADA)
%MX290	UP201B    Run  (SCADA)
%MX291	UP201B   Stop  (SCADA)
%MX294	UP202A    Run  (SCADA)
%MX295	UP202A   Stop  (SCADA)
%MX298	UP202B    Run  (SCADA)
%MX299	UP202B   Stop  (SCADA)
%MX302	UP203A    Run  (SCADA)
%MX303	UP203A   Stop  (SCADA)
%MX306	UP203B    Run  (SCADA)
%MX307	UP203B   Stop  (SCADA)
%MX310	TANK101 Level 95%   HH
%MX312	TK-101 ATG Trouble
%MX314	TANK101 Level 10%   LL
%MX320	TANK102 Level 95%   HH
%MX322	TK-102 ATG Trouble
%MX324	TANK102 Level 10%   LL
%MX330	TANK103 Level 95%   HH
%MX332	TK-103 ATG Trouble
%MX334	TANK103 Level 10%   LL
%MX340	TANK104 Level 95%   HH
%MX342	TK-104 ATG Trouble
%MX344	TANK104 Level 10%   LL
%MX350	TANK105 Level 95%   HH
%MX352	TK-105 ATG Trouble
%MX354	TANK105 Level 10%   LL
%MX360	TANK106 Level 95%   HH
%MX362	TK-106 ATG Trouble
%MX364	TANK106 Level 10%   LL
%MX370	TANK107 Level 95%   HH
%MX372	TK-107 ATG Trouble
%MX374	TANK107 Level 10%   LL
%MX380	TANK108 Level 95%   HH
%MX382	TK-108 ATG Trouble
%MX384	TANK108 Level 10%   LL
%MX390	TANK109 Level 95%   HH
%MX392	TK-109 ATG Trouble
%MX394	TANK109 Level 10%   LL
%MX400	TANK110 Level 95%   HH
%MX402	TK-110 ATG Trouble
%MX404	TANK110 Level 10%   LL
%MX410	TANK111 LEVEL 95% HH
%MX411	TANK111 Level 90% H
%MX413	TANK Level 15% L
%MX414	TANK111 Level 10% LL
%MX420	TANK112 LEVEL 95% HH
%MX421	TANK112 LEVEL 90% H
%MX423	TANK112 LEVEL 15% L
%MX424	TANK112 LEVEL 10% LL
%MX430	TANK113 LEVEL 95% HH
%MX431	TANK113 LEVEL 90% H
%MX433	TANK113 LEVEL 15% L
%MX434	TANK113 LEVEL 10% LL
%MX448	P101A Auto 1차 운전 선택 Switch(SCADA)
%MX449	P101B Auto 1차 운전 선택 Switch(SCADA)
%MX450	P102A Auto 1차 운전 선택 Switch(SCADA)
%MX451	P102B Auto 1차 운전 선택 Switch(SCADA)
%MX452	P103A Auto 1차 운전 선택 Switch(SCADA)
%MX453	P103B Auto 1차 운전 선택 Switch(SCADA)
%MX454	P104A Auto 1차 운전 선택 Switch(SCADA)
%MX455	P104B Auto 1차 운전 선택 Switch(SCADA)
%MX456	P107A Auto 1차 운전 선택 Switch(SCADA)
%MX457	P107B Auto 1차 운전 선택 Switch(SCADA)
%MX458	P108A Auto 1차 운전 선택 Switch(SCADA)
%MX459	P108B Auto 1차 운전 선택 Switch(SCADA)
%MX460	P101A Auto 2차 운전 선택 Switch(SCADA)
%MX461	P101B Auto 2차 운전 선택 Switch(SCADA)
%MX462	P102A Auto 2차 운전 선택 Switch(SCADA)
%MX463	P102B Auto 2차 운전 선택 Switch(SCADA)
%MX464	P103A Auto 2차 운전 선택 Switch(SCADA)
%MX465	P103B Auto 2차 운전 선택 Switch(SCADA)
%MX466	P104A Auto 2차 운전 선택 Switch(SCADA)
%MX467	P104B Auto 2차 운전 선택 Switch(SCADA)
%MX468	P107A Auto 2차 운전 선택 Switch(SCADA)
%MX469	P107B Auto 2차 운전 선택 Switch(SCADA)
%MX470	P108A Auto 2차 운전 선택 Switch(SCADA)
%MX472	Auto 선택 완료    (SCADA)
%MX473	Q/T Alarm
%MX474	120대대 Alarm
%MX475	121대대 Alarm
%MX476	123대대 Alarm
%MX477	157대대 Alarm
%MX478	HS Alarm
%MX479	HS 이송 MOV
%MX500	통신 읽기 PULS1
%MX501	통신 읽기 PULS2
%MX502	통신 읽기 PULS3
%MX503	통신 읽기 PULS4
%MX504	통신 읽기 PULS5
%MX505	통신 읽기 PULS RESET
%MX513	HLV20301 TK101 Open SIG(MANU)
%MX514	HLV20301 TK101 Open SIG(Auto)
%MX516	HLV20301 TK102 Open SIG(MANU)
%MX517	HLV20301 TK102 Open SIG(Auto)
%MX519	HLV20501 TK103 Open SIG(MANU)
%MX520	HLV20501 TK103 Open SIG(Auto)
%MX522	HLV20601 TK104 Open SIG(MANU)
%MX523	HLV20601 TK104 Open SIG(Auto)
%MX525	HLV20901 TK107 Open SIG(MANU)
%MX526	HLV20901 TK107 Open SIG(Auto)
%MX528	HLV21001 TK108 Open SIG(MANU)
%MX529	HLV21001 TK108 Open SIG(Auto)
%MX530	HLV20701 TK105 Open PULS(MANU)
%MX531	HLV20701 TK105 Open SIG
%MX532	HLV20801 TK106 Open PULS(MANU)
%MX533	HLV20801 TK106 Open SIG
%MX534	HLV21101 TK109 Open PULS(MANU)
%MX535	HLV21101 TK109 Open SIG
%MX536	HLV21201 TK110 Open PULS(MANU)
%MX537	HLV21201 TK110 Open SIG
%MX700	TK-111 HH or HLVD Trouble
%MX701	TK-112 HH or HLVD Trouble
%MX702	TK-113 HH or HLVD Trouble
%MX704	ARES 공통 정지 조건
%MX705	HH Stop Logic
(TK101)
%MX706	HH Stop Logic
(TK102)
%MX707	HH Stop Logic
(TK103)
%MX708	HH Stop Logic
(TK104)
%MX709	HH Stop Logic
(TK105)
%MX710	HH Stop Logic
(TK106)
%MX711	HH Stop Logic
(TK107)
%MX712	HH Stop Logic
(TK108)
%MX713	ARES SUMP 공통 정지 조건
%MX714	JP-8
[#5,#6]
공통 정지조건
%MX715	JP-8 SUMP
[#5,#6]
공통 정지조건
%MX716	DIESEL
[#9,#10]
공통 정지조건
%MX717	DIESEL SUMP
[#9,#10]
공통 정지조건
%MX718	HH Stop Logic
(TK109)
%MX719	HH Stop Logic
(TK110)
%MX810	TK-101 HH SIG
%MX811	TK101 H SIG
%MX813	TK101 L SIG
%MX814	TK-101 LL SIG
%MX820	TK-102 HH SIG
%MX821	TK102 H SIG
%MX823	TK102 L SIG
%MX824	TK-102 LL SIG
%MX830	TK-103 HH SIG
%MX831	TK103 H SIG
%MX833	TK103 L SIG
%MX834	TK-103 LL SIG
%MX840	TK-104 HH SIG
%MX841	TK104 H SIG
%MX843	TK104 L SIG
%MX844	TK-104 LL SIG
%MX850	TK-105 HH SIG
%MX851	TK105 H SIG
%MX853	TK105 L SIG
%MX854	TK-105 LL SIG
%MX860	TK-106 HH SIG
%MX861	TK106 H SIG
%MX863	TK106 L SIG
%MX864	TK-106 LL SIG
%MX870	TK-107 HH SIG
%MX871	TK107 H SIG
%MX873	TK107 L SIG
%MX874	TK-107 LL SIG
%MX880	TK-108 HH SIG
%MX881	TK108 H SIG
%MX883	TK108 L SIG
%MX884	TK-108 LL SIG
%MX890	TK-109 HH SIG
%MX891	TK109 H SIG
%MX893	TK109 L SIG
%MX894	TK-108 LL SIG
%MX900	TK-110 HH SIG
%MX901	TK110 H SIG
%MX903	TK110 L SIG
%MX904	TK-110 LL SIG
%MX910	TK-111 HH SIG
%MX911	TK-111 H SIG
%MX913	TK-111 L SIG
%MX914	TK-111 LL SIG
%MX920	TK-112 HH SIG
%MX921	TK-112 H SIG
%MX923	TK-112 L SIG
%MX924	TK-112 LL SIG
%MX930	TK-113 HH SIG
%MX931	TK-113 H SIG
%MX933	TK-113 L SIG
%MX934	TK-113 LL SIG
%MX6400	Panel Manual
%MX6401	SCADA Manual
%MX6402	Panel  Auto
%MX6403	SCADA  Auto
%MX6404	TOTAL Emergency
%MX6405	BUZZER Stop
%MX6406	TOTAL Alarm
%MX6409	SQ_EM (ARES Stop)
%MX6410	Manual 선택
%MX6411	Auto 선택
%MX6412	JP-8 
#5, #6 Alarm
%MX6413	DIESEL
#9, #10
Alarm
%MX6414	SQ 120 EM (ARES STOP)
%MX6415	SQ 121 EM (ARES STOP)
%MX6416	SQ 123 EM (ARES STOP)
%MX6417	SQ 157 EM (ARES STOP)
%MX6419	Power on 보조
[SCADA]
%MX6420	POL Alarm
%MX6421	TK-101 HH & HLV OPEN
%MX6422	TK-102 HH & HLV OPEN
%MX6423	TK-103 HH & HLV OPEN
%MX6424	TK-104 HH & HLV OPEN
%MX6425	ARES 
Alarm
%MX6427	TK-107 HH & HLV OPEN
%MX6428	TK-108 HH & HLV OPEN
%MX6430	QT, HS, SQ Alarm
%MX6431	TK-105 HH & HLV OPEN
%MX6432	TK-106 HH & HLV OPEN
%MX6433	TK-109 HH & HLV OPEN
%MX6434	TK-110 HH & HLV OPEN
%MX6435	Horn Stop Reset
%MX6464	Lamp Test SIG
%MX6465	TK101-EM
%MX6466	TK102-EM
%MX6467	TK103-EM
%MX6468	TK104-EM
%MX6469	TK105-EM
%MX6470	TK106-EM
%MX6471	TK107-EM
%MX6472	TK108-EM
%MX6473	TK109-EM
%MX6474	TK110-EM
%MX6475	PUMP실-EM 
%MX6476	MAIN PNL-EM
%MX6477	LDS PNL EM
%MX6478	TK-108 LEAK Alarm
%MX6479	PANTO1_EM
%MX6480	PANTO2_EM
%MX6481	PANTO3_EM
%MX6482	PANTO4_EM
%MX6483	PANTO5_EM
%MX7042	ARES_EM
%MX7043	JP-8
#5, #6
Emergency
%MX7044	DIESEL
#9, #10
Emergency
%MX13440	P110A Run SIG
%MX13441	P110B Run SIG
%MX13442	P110C Run SIG
%MX13443	DRAIN TK-111 Run SIG
%MX13444	DRAIN TK-112 Run SIG
%MX13445	DRAIN TK-113 Run SIG
%MX13446	MOV20103 수동 Open
%MX13447	MOV20103 수동 Close
%MX13448	MOV20104 수동 Open
%MX13449	MOV20104 수동 Close
%MX13450	MOV20102 수동 Open
%MX13451	MOV20102 수동 Close
%MX13452	MOV20105 수동 Open
%MX13453	MOV20105 수동 Close
%MX13454	MOV20101 수동 Open
%MX13455	MOV20101 수동 Close
%MX13456	UP201A Run SIG
%MX13457	UP201B Run SIG
%MX13458	UP202A Run SIG
%MX13459	UP202B Run SIG
%MX13460	UP203A Run SIG
%MX13461	UP203B Run SIG
%MX14081	TK-101 수령 SIG [SCADA -> PLC]
%MX14082	TK-102 수령 SIG [SCADA -> PLC]
%MX14083	TK-103 수령 SIG [SCADA -> PLC]
%MX14084	TK-104 수령 SIG [SCADA -> PLC]
%MX14087	TK-107 수령 SIG [SCADA -> PLC]
%MX14088	TK-108 수령 SIG [SCADA -> PLC]
%MX19200	P101A Alarm
%MX19201	P101A FS Alarm
%MX19204	P101B Alarm
%MX19205	P101B FS Alarm
%MX19208	P101C Alarm
%MX19209	P101C FS Alarm
%MX19212	P102A Alarm
%MX19213	P102A FS Alarm
%MX19216	P102B Alarm
%MX19217	P102B FS Alarm
%MX19220	P102C Alarm
%MX19221	P102C FS Alarm
%MX19224	P103A Alarm
%MX19225	P103A FS Alarm
%MX19228	P103B Alarm
%MX19229	P103B FS Alarm
%MX19232	P103C Alarm
%MX19233	P103C FS Alarm
%MX19236	P104A Alarm
%MX19237	P104A FS Alarm
%MX19240	P104B Alarm
%MX19241	P104B FS Alarm
%MX19244	P104C Alarm
%MX19245	P104C FS Alarm
%MX19248	P105A Alarm
%MX19249	P105A FS Alarm
%MX19252	P105B Alarm
%MX19253	P105B FS Alarm
%MX19264	P101A Run SIG
%MX19265	P101B Run SIG
%MX19266	P101C Run SIG
%MX19267	P101A Lock key Run
%MX19268	P101B Lock key Run
%MX19269	P101C Lock key Run
%MX19270	P102A Lock key Run
%MX19271	P102B Lock key Run
%MX19272	P102C Lock key Run
%MX19273	P103A Lock key Run
%MX19274	P103B Lock key Run
%MX19275	P103C Lock key Run
%MX19276	P104A Lock key Run
%MX19277	P104B Lock key Run
%MX19278	P104C Lock key Run
%MX19279	P105A Lock key Run
%MX19280	P105B Lock key Run
%MX19281	P105C Lock key Run
%MX19282	P106A Lock key Run
%MX19283	P106B Lock key Run
%MX19284	P106C Lock key Run
%MX19285	P107A Lock key Run
%MX19286	P107B Lock key Run
%MX19287	P107C Lock key Run
%MX19288	P108A Lock key Run
%MX19289	P108B Lock key Run
%MX19290	P108C Lock key Run
%MX19291	P109A Lock key Run
%MX19292	P109B Lock key Run
%MX19293	P109C Lock key Run
%MX19294	P110A Lock key Run
%MX19295	P110B Lock key Run
%MX19296	P110C Lock key Run
%MX19297	P111 Lock key Run
%MX19298	P112 Lock key Run
%MX19299	P113 Lock key Run
%MX19328	P102A Run SIG
%MX19329	P102B Run SIG
%MX19330	P102C Run SIG
%MX19392	P103A Run SIG
%MX19393	P103B Run SIG
%MX19394	P103C Run SIG
%MX19456	P104A Run SIG
%MX19457	P104B Run SIG
%MX19458	P104C Run SIG
%MX19520	P105A Run SIG
%MX19521	P105B Run SIG
%MX19522	P105C Run SIG
%MX19584	P106A Run SIG
%MX19585	P106B Run SIG
%MX19586	P106C Run SIG
%MX19648	P107A Run SIG
%MX19649	P107B Run SIG
%MX19650	P107C Run SIG
%MX19712	P108A Run SIG
%MX19713	P108B Run SIG
%MX19714	P108C Run SIG
%MX19776	P109A Run SIG
%MX19777	P109B Run SIG
%MX19778	P109C Run SIG
%MX19840	P105C Alarm
%MX19841	P105C FS Alarm
%MX19844	P106A Alarm
%MX19845	P106A FS Alarm
%MX19847	P106B Alarm
%MX19848	P106B FS Alarm
%MX19851	P106C Alarm
%MX19852	P106C FS Alarm
%MX19855	P107A Alarm
%MX19856	P107A FS Alarm
%MX19859	P107B Alarm
%MX19860	P107B FS Alarm
%MX19863	P107C Alarm
%MX19864	P107C FS Alarm
%MX19867	P108A Alarm
%MX19868	P108A FS Alarm
%MX19871	P108B Alarm
%MX19872	P108B FS Alarm
%MX19875	P108C Alarm
%MX19876	P108C FS Alarm
%MX19879	P109A Alarm
%MX19880	P109A FS Alarm
%MX19883	P109B Alarm
%MX19884	P109B FS Alarm
%MX19887	P109C Alarm
%MX19888	P109C FS Alarm
%MX19891	P110A Alarm
%MX19892	P110A FS Alarm
%MX19895	P110B Alarm
%MX19896	P110B FS Alarm
%MX19899	P110C Alarm
%MX19900	P110C FS Alarm
%MX19903	TK-111 Alarm
%MX19904	TK-111 FS Alarm
%MX19907	TK-112 Alarm
%MX19908	TK-112 FS Alarm
%MX19911	TK-113 Alarm
%MX19912	TK-113 FS Alarm
%MX19913	UP201A Alarm
%MX19914	UP201B Alarm
%MX19915	UP202A Alarm
%MX19916	UP202B Alarm
%MX19917	UP203A Alarm
%MX19918	UP203B Alarm
%MX19919	UP201A FS Alarm
%MX19920	UP201B FS Alarm
%MX19921	UP202A FS Alarm
%MX19922	UP202B FS Alarm
%MX19923	UP203A FS Alarm
%MX19924	UP203B FS Alarm
%MX20544	60sec 주기 CLock
%MX20545	60min 주기 CLock
%MX21120	P101A FS SIG
%MX21121	P101B FS SIG
%MX21122	P101C FS SIG
%MX21123	P102A FS SIG
%MX21124	P102B FS SIG
%MX21125	P102C FS SIG
%MX21126	P103A FS SIG
%MX21127	P103B FS SIG
%MX21128	P103C FS SIG
%MX21129	P104A FS SIG
%MX21130	P104B FS SIG
%MX21131	P104C FS SIG
%MX21132	P105A FS SIG
%MX21133	P105B FS SIG
%MX21134	P105C FS SIG
%MX21135	P106A FS SIG
%MX21136	P106B FS SIG
%MX21137	P106C FS SIG
%MX21138	P107A FS SIG
%MX21139	P107B FS SIG
%MX21140	P107C FS SIG
%MX21141	P108A FS SIG
%MX21142	P108B FS SIG
%MX21143	P108C FS SIG
%MX21144	P109A FS SIG
%MX21145	P109B FS SIG
%MX21146	P109C FS SIG
%MX21147	P110A FS SIG
%MX21148	P110B FS SIG
%MX21149	P110C FS SIG
%MX21150	P111 FS SIG
%MX21151	P112 FS SIG
%MX21152	P113 FS SIG
%MX21153	ARES LOOP Stop (SCADA => PLC)
%MX21154	UP201A FS SIG
%MX21155	UP201B FS SIG
%MX21156	UP202A FS SIG
%MX21157	UP202B FS SIG
%MX21158	UP203A FS SIG
%MX21159	UP203B FS SIG
%MX21160	ARES TANK HH & HLV OPEN
%MX21161	JP-8 TK #5, #6 HH & HLV OPEN
%MX21162	DIESEL TANK HH & HLV OPEN
%MX23040	수령선택 RESET
%MX23041	수령선택 TK-101
%MX23042	수령선택 TK-102
%MX23043	수령선택 TK-103
%MX23044	수령선택 TK-104
%MX23047	수령선택 TK-107
%MX23048	수령선택 TK-108 [SCADA -> PLC]
%MX23078	ARES LOOP Stop
%MX23080	ARES LOOP Stop RESET
%MX23081	ARES (HLV All Close SIG)
%MX23082	ARES HLV All Close SIG
%MX23083	JP-8 TK #5, #6 HLV All Close SIG
%MX23085	Diesel TK #9, #10 HLV All Close SIG
%MX23087	Auto start all ready
%MX23089	ARES Stop SIG
%MX23681	TANK 101 수령 송유관 색변화
%MX23682	TANK 102 수령 송유관 색변화
%MX23683	TANK 103 수령 송유관 색변화
%MX23684	TANK 104 수령 송유관 색변화
%MX23685	TANK 107 수령 송유관 색변화
%MX23686	TANK 108 수령 송유관 색변화
%MX23692	TANK 105 수령 송유관 색변화
%MX23693	TANK 105,106 공통 불출 송유관 색변화
%MX23695	TANK 106 수령 송유관 색변화
%MX23704	TANK 109 수령 송유관 색변화
%MX23705	TANK 109,110 공통 불출 송유관 색변화
%MX23707	TANK 110 수령 송유관 색변화
%MX23716	회수 송유관 색변화 MAIN LINE
%MX25600	Auto Start OK
%MX25601	Auto Start SIG
%MX25602	All Remote
%MX25664	P101A Auto 1차 Run
%MX25665	P101A Auto 2차 Run
%MX25666	P101B Auto 1차 Run
%MX25667	P101B Auto 2차 Run
%MX25728	P102A Auto 1차 Run
%MX25729	P102A Auto 2차 Run
%MX25730	P102B Auto 1차 Run
%MX25731	P102B Auto 2차 Run
%MX25792	P103A Auto 1차 Run
%MX25793	P103A Auto 2차 Run
%MX25794	P103B Auto 1차 Run
%MX25795	P103B Auto 2차 Run
%MX25856	P104A Auto 1차 Run
%MX25857	P104A Auto 2차 Run
%MX25858	P104B Auto 1차 Run
%MX25859	P104B Auto 2차 Run
%MX25920	P107A Auto 1차 Run
%MX25921	P107A Auto 2차 Run
%MX25922	P107B Auto 1차 Run
%MX25923	P107B Auto 2차 Run
%MX25984	P108A Auto 1차 Run
%MX25985	P108A Auto 2차 Run
%MX25986	P108B Auto 1차 Run
%MX25987	P108B Auto 2차 Run
%MX26112	Auto 2st 
Pump Run
%MX26113	TLV Count >= Zero
%MX26176	mov 107 return open
%MX26177	mov 107 return close
%MX26178	MOV20102 Open
%MX26179	MOV20102
Close
%MX26240	1차 펌프 Running Timing
%MX26241	2차 펌프 Running Timing
%MX26242	1차 PUMP Stoping Timing
%MX26243	2차 PUMP Stoping Timing
%MX26244	Auto BPCV Stop
%MX26246	1차 펌프 정지조건 홀딩
%MX26266	Auto CVP stop
%WW1	HLV20301 TK101 SET
%WW2	HLV20301 TK102 SET
%WW3	HLV20501 TK103 SET
%WW4	HLV20601 TK104 SET
%WW7	HLV20901 TK107 SET
%WW8	HLV21001 TK108 SET
%WW9	To HS 
[16 BIT]
%WW10	TK-101 ATG TROUBLE
%WW11	출하 PUMP 2차 운전 선택 SET
%WW13	 P302 2차 선택 SET
%WW20	TANK101 문자열
%WW21	TANK102 문자열
%WW22	TANK103 문자열
%WW23	TANK104 문자열
%WW24	TANK105 문자열
%WW25	TANK106 문자열
%WW26	TANK107문자열
%WW27	TANK108 문자열
%WW28	TANK109 문자열
%WW29	TANK110 문자열
%WW110	출하 PUMP 1차 운전 선택 SET
%WW120	출하PUMP 2차 운전선택 SET
%WW150	P101A Run SET
%WW151	P101B Run SET
%WW152	P101C Run SET
%WW153	P102A Run SET
%WW154	P102B Run SET
%WW155	P102C Run SET
%WW156	P103A Run SET
%WW157	P103B Run SET
%WW158	P103C Run SET
%WW159	P104A Run SET
%WW160	P104B Run SET
%WW161	P104C Run SET
%WW162	P105A Run SET
%WW163	P105B Run SET
%WW164	P105C Run SET
%WW165	P106A Run SET
%WW166	P106B Run SET
%WW167	P106C Run SET
%WW168	P107A Run SET
%WW169	P107B Run SET
%WW170	P107C Run SET
%WW171	P108A Run SET
%WW172	P108B Run SET
%WW173	P108C Run SET
%WW174	P109A Run SET
%WW175	P109B Run SET
%WW176	P109C Run SET
%WW177	P110A Run SET
%WW178	P110B Run SET
%WW179	P110C Run SET
%WW180	DRAIN TK-111 Run SET
%WW181	DRAIN TK112 Run SET
%WW182	DRAIN TK113 Run SET
%WW183	MOV 20103 Open SET
%WW184	MOV 20104 Open SET
%WW185	MOV 20102 Open SET
%WW186	MOV 20105 Open SET
%WW187	MOV 20101 Open SET
%WW188	ARES UP201A Run SET
%WW189	ARES UP201B Run SET
%WW190	Diesel UP202A Run SET
%WW191	Diesel UP202B Run SET
%WW192	TANK#5,6 UP203A Run SET
%WW193	TANK#5,6 UP203B Run SET
%WW250	초단위
%WW251	분단위
%WW252	시단위
%WW401	401TK Level
%WW402	402TK Level
%WW403	403TK Level
%WW404	404TK Level
%WW410	PT101 회수압력
%WW412	PT101 회수압력계 레인지 연산값
%WW416	PT101 회수압력 x 10
%WW420	PT102 불출압력
%WW422	PT102 불출압력계 레인지 연산값
%WW426	PT102 불출압력 x10
%WW430	FT101 불출유량
%WW432	FT103 회수유량계 레인지 연산값
%WW436	FT101 불출유량 x10
%WW440	FT103 회수유량
%WW442	FT103 회수유량계 레인지 연산값
%WW446	FT103 회수유량 x10
%WW500	TK-111 Level 변환값
%WW506	DRAIN TANK TK-111 Level (PLC => SCADA)
%WW510	TK-112 Level 변환값
%WW516	DRAIN TANK 112 Level (PLC => SCADA()
%WW520	DRAIN TANK 113 변환값
%WW526	DRAIN TANK TK-113 Level (PLC => SCADA)
%WW530	아날로그입력 모듈: 채널7 변환값
%WW602	TK101 Volume(CATAMS=>PLC)
%WW603	TK101 Volume(CATAMS=>PLC)
%WW606	TK102 Volume(CATAMS=>PLC)
%WW607	TK102 Volume(CATAMS=>PLC)
%WW610	TK103 Volume(CATAMS=>PLC)
%WW611	TK103 Volume(CATAMS=>PLC)
%WW614	TK104 Volume(CATAMS=>PLC)
%WW615	TK104 Volume(CATAMS=>PLC)
%WW618	TK105 Volume(CATAMS=>PLC)
%WW619	TK105 Volume(CATAMS=>PLC)
%WW622	TK106 Volume(CATAMS=>PLC)
%WW623	TK106 Volume(CATAMS=>PLC)
%WW626	TK107 Volume(CATAMS=>PLC)
%WW627	TK107 Volume(CATAMS=>PLC)
%WW630	TK108 Volume(CATAMS=>PLC)
%WW631	TK108 Volume(CATAMS=>PLC)
%WW634	TK109 Volume(CATAMS=>PLC)
%WW635	TK109 Volume(CATAMS=>PLC)
%WW638	TK110 Volume(CATAMS=>PLC)
%WW639	TK110 Volume(CATAMS=>PLC)
%WW642	TK111 Volume(CATAMS=>PLC)
%WW643	TK111 Volume(CATAMS=>PLC)
%WW646	TK112 Volume(CATAMS=>PLC)
%WW647	TK112 Volume(CATAMS=>PLC)
%WW650	TK113 Volume(CATAMS=>PLC)
%WW651	TK113 Volume(CATAMS=>PLC)
%WW654	401 Volume CATAMS => PLC
%WW655	401 Volume CATAMS => PLC
%WW658	402 Volume CATAMS =>PLC
%WW659	402 Volume CATAM => PLC
%WW662	403 Volume CATAMS => PLC
%WW663	403 Volume CATAMS => PLC
%WW666	404 Volume CATAMS => PLC
%WW667	404 Volume CATAMS => PLC
%WW670	TK-001 Volume (CTM=>POL)
%WW671	TK-001 Volume (CTM=>POL)
%WW674	TK-002 Volume(CTM => POL)
%WW675	TK-002 Volume (CTM => POL)
%WW678	TK-003 Volume (CTM => POL)
%WW679	TK-003 Volume (CTM => POL)
%WW682	TK-301 Volume (CTM => POL)
%WW683	TK-301 Volume (CTM => POL)
%WW686	TK-302 Volume (CTM => POL)
%WW687	TK-302 Volume (CTM => POL)
%WW690	TK-303 Volume (CTM => POL)
%WW691	TK-303 Volume (CTM => POL)
%WW900	TK-101   Level
From.NMR#1
%WW901	TK-101 ATG TROUBLE
From.NMR#1
%WW903	TK-102 Level
From.NMR#1
%WW904	TK-102 ATG TROUBLE
From.NMR#1
%WW906	TK-103 Level
From.NMR#1
%WW907	TK-103 ATG TROUBLE
From.NMR#1
%WW909	TK-104 Level
From.NMR#1
%WW910	TK-104 ATG TROUBLE
From.NMR#1
%WW912	TK-105 Level
From.NMR#1
%WW913	TK-105 ATG TROUBLE
From.NMR#1
%WW915	TK-106 Level
From.NMR#1
%WW916	TK-106 ATG TROUBLE
From.NMR#1
%WW918	TK-107 Level
From.NMR#1
%WW919	TK-107 ATG TROUBLE
From.NMR#1
%WW921	TK-108 Level
From.NMR#1
%WW922	TK-108 ATG TROUBLE
From.NMR#1
%WW924	TK-109 Level
From.NMR#1
%WW925	TK-109 ATG TROUBLE
From.NMR#1
%WW927	TK-110 Level
From.NMR#1
%WW928	TK-110 ATG TROUBLE
From.NMR#1
%WW1001	TK-101   Level  (CTM=>PLC)
%WW1100	DRAIN TANK 111 => NMR5000
%WW1103	DRAIN TANK 112 => NMR5000
%WW1106	DRAIN TANK 113 => NMR5000
%WW1109	DRAIN TANK 401 => NMR5000
%WW1112	DRAIN TANK 402 => NMR5000
%WW1115	DRAIN TANK 403 => NMR5000
%WW1118	DRAIN TANK 404 => NMR5000
%WW1600	SQ_TLV_COUNT
%WW4001	TK-101   Level
From.NMR#1
%WW4002	TK-101 ATG TROUBLE
From.NMR#1
%WW4004	TK-102 Level
From.NMR#1
%WW4005	TK-102 ATG TROUBLE
From.NMR#1
%WW4007	TK-103 Level
From.NMR#1
%WW4008	TK-103 ATG TROUBLE
From.NMR#1
%WW4010	TK-104 Level
From.NMR#1
%WW4011	TK-104 ATG TROUBLE
From.NMR#1
%WW4013	TK-105 Level
From.NMR#1
%WW4014	TK-105 ATG TROUBLE
From.NMR#1
%WW4016	TK-106 Level
From.NMR#1
%WW4017	TK-106 ATG TROUBLE
From.NMR#1
%WW4019	TK-107 Level
From.NMR#1
%WW4020	TK-107 ATG TROUBLE
From.NMR#1
%WW4022	TK-108 Level
From.NMR#1
%WW4023	TK-108 ATG TROUBLE
From.NMR#1
%WW4025	TK-109 Level
From.NMR#1
%WW4026	TK-109 ATG TROUBLE
From.NMR#1
%WW4028	TK-110 Level
From.NMR#1
%WW4029	TK-110 ATG TROUBLE
From.NMR#1
%WD412	PT101 회수압력계 레인지 연산값 2WORD 변환
%WD414	PT101 회수압력 연산값
%WD416	PT101 회수압력 2WORD 변환
%WD418	PT101 회수압력 보정값
%WD422	PT102 불출압력계 레인지 연산값 2WORD 변환
%WD424	PT102 불출압력 연산값
%WD426	PT102 불출압력 2WORD 변환
%WD428	PT102 불출압력 보정값
%WD432	FT101 불출유량계 레인지 연산값 2WORD 변환
%WD434	FT101 불출유량 연산값
%WD436	FT101 불출유량 2WORD 변환
%WD438	FT101 불출유량 보정값
%WD440	불출유량 - 회수유량 = 값
%WD442	FT103 회수유량계 레인지 연산값 2WORD 변환
%WD444	FT103 회수유량 연산값
%WD446	FT103 회수유량 2WORD 변환
%WD448	FT103 회수유량 보정값
%WD500	TK-111 Level 변환값(wd)
%WD504	DRAIN TANK 111 Volume
%WD510	TK-112 Level 변환값(wd)
%WD514	DRAIN TANK 112 Volume
%WD520	TK-113 Level 변환값(WD)
%WD524	DRAIN TANK 113 Volume
%WD560	TANK 101,102 Volume 합산
%WD562	TANK 103,104 Volume 합산
%WD564	TANK 105,106 Volume 합산
%WD566	TANK 107,108 Volume 합산
%WD570	TANK 101,102, 103,104 Volume 합산
%WD580	TANK 105,106, 107,108 Volume 합산
%WD590	TANK Volume 합산
%WD654	401 PLC => SCADA Volume
%WD658	402 Volume PLC => SCADA
%WD662	403 Volume PLC => SCADA
%WD666	404 Volume PLC => SCADA
%WD670	TK-001 Volume (POL => SCADA)
%WD674	TK-002 Volume (POL => SCADA)
%WD678	TK-003 Volume (POL => SCADA)
%WD682	TK-301 Volume (POL => SCADA)
%WD686	TK-302 Volume (POL => SCADA)
%WD690	TK-303 Volume (POL => SCADA)
%WD700	TK-101 Level Height
%WD708	TANK 101 Volume
%WD710	TK-102 Level Height
%WD718	TANK 102 Volume
%WD720	TK-103 Level Height
%WD728	TANK 103 Volume
%WD730	TK-104 Level Height
%WD738	TANK 104 Volume
%WD740	TK-105 Level Height
%WD748	TANK 105 Volume
%WD750	TK-106 Level Height
%WD758	TANK 106 Volume
%WD760	TK-107 Level Height
%WD768	TANK 107 Volume
%WD770	TK-108 Level Height
%WD778	TANK 108 Volume
%WD780	TK-109 Level Height
%WD788	TANK 109 Volume
%WD790	TK-110 Level Height
%WD798	TANK 110 Volume
*)

PROGRAM Main (* task: 스캔 프로그램 *)
VAR
    AUTO_S_FS : TON;
    BPCV_OFF : TOF; (* BPCV OFF DELAY *)
    CVP : TON;
    CVP_OFF : TOF; (* CVP OFF DELAY *)
    CVP_OFF1 : TOF; (* CVP OFF DELAY *)
    CVP_OFF_DELAY : TOF;
    INST : CTD_DINT;
    INST1 : TOF;
    LDS_ALARM : TON;
    L_TST : TON;
    L_TST1 : TON;
    L_TST_FS : TON;
    L_TST_FS1 : TON;
    P101A_FS : TON; (* P101A_FS Alarm TON *)
    TP19 : TP; (* P107 FS 30초 Holdding *)
END_VAR
VAR_EXTERNAL
    _0100_CH3_DATA : INT; (* AT %UW1.0.5 *) (* 아날로그입력 모듈: 채널3 변환값 *)
END_VAR
VAR
    _e1 : R_TRIG;
    _e2 : R_TRIG;
    _e3 : R_TRIG;
    _e4 : R_TRIG;
    _e5 : R_TRIG;
END_VAR

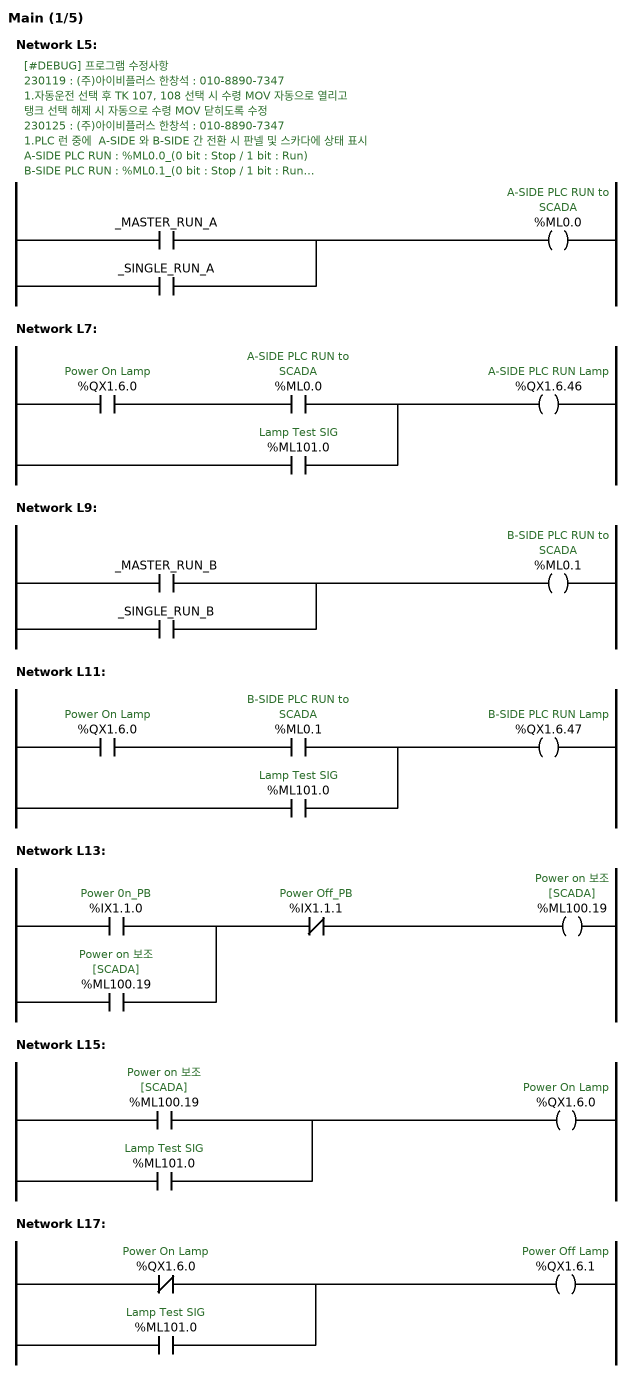
(* [#DEBUG] 프로그램 수정사항 *)
(* 230119 : (주)아이비플러스 한창석 : 010-8890-7347 / 1.자동운전 선택 후 TK 107, 108 선택 시 수령 MOV 자동으로 열리고 / 탱크 선택 해제 시 자동으로 수령 MOV 닫히도록 수정 *)
(* 230125 : (주)아이비플러스 한창석 : 010-8890-7347 / 1.PLC 런 중에  A-SIDE 와 B-SIDE 간 전환 시 판넬 및 스카다에 상태 표시 / A-SIDE PLC RUN : %ML0.0_(0 bit : Stop / 1 bit : Run) / B-SIDE PLC RUN : %ML0.1_(0 bit : Stop / 1 bit : Run) / 2.ATG 각 상태 (HH,H,L,LL) 별 알림창 과 부저 발생 상황 정리 / - HH 발생시 그 탱크 외 해당 탱크와 연관 된 다른 탱크의 불출 펌프 / 모두 정지 및 부저 발생. / - HH 발생시 스카다에 발생한 탱크의 상태 및 알림창 팝업. / - H 발생시 스카다에 발생한 탱크의 상태 및 알림창 팝업. / - L 발생시 스카다에 발생한 탱크의 상태 및 알림창 팝업. / - LL 발생시 발생한 탱크의 불출펌프 정지 및 부저 발생. / - LL 발생시 스카다에 발생한 탱크의 상태 및 알림창 팝업. / - Drain tank HH 발생시 해당 드레인탱크와 연관 된 다른 탱크의 Sump pump / 모두 정지. / 3.ATG 통신이상 발생시 개별적인지 통합이상인지 판단하여 스카다에 표시 및 / 해당 상황에 맞추어 스카다 제어를 제한하고 판넬 및 현장 제어만 가능하도록 한다. / 4.OCR 및 기타 개별 펌프관련 이상 발생시 판넬 트러블 표시램프 점등 후 상태를 / 유지하고 문제 해결 후 스카다 또는 판넬에서 RESET버튼으로 해제 가능하도록 수정. *)
(* 230205 : 각 탱크별 유위 알람 설정치를 보기 쉽도록 ST언어로 변경하여 프로그램 *)
(* /////// CONTROL /////// *)
(* Rung L5 *)
%ML0.0 := _MASTER_RUN_A OR _SINGLE_RUN_A;
(* Rung L7 *)
%QX1.6.46 := (%QX1.6.0 AND %ML0.0) OR %ML101.0;
(* Rung L9 *)
%ML0.1 := _MASTER_RUN_B OR _SINGLE_RUN_B;
(* Rung L11 *)
%QX1.6.47 := (%QX1.6.0 AND %ML0.1) OR %ML101.0;
(* Rung L13 *)
%ML100.19 := (%IX1.1.0 OR %ML100.19) AND NOT %IX1.1.1;
(* Rung L15 *)
%QX1.6.0 := %ML100.19 OR %ML101.0;
(* Rung L17 *)
%QX1.6.1 := NOT %QX1.6.0 OR %ML101.0;

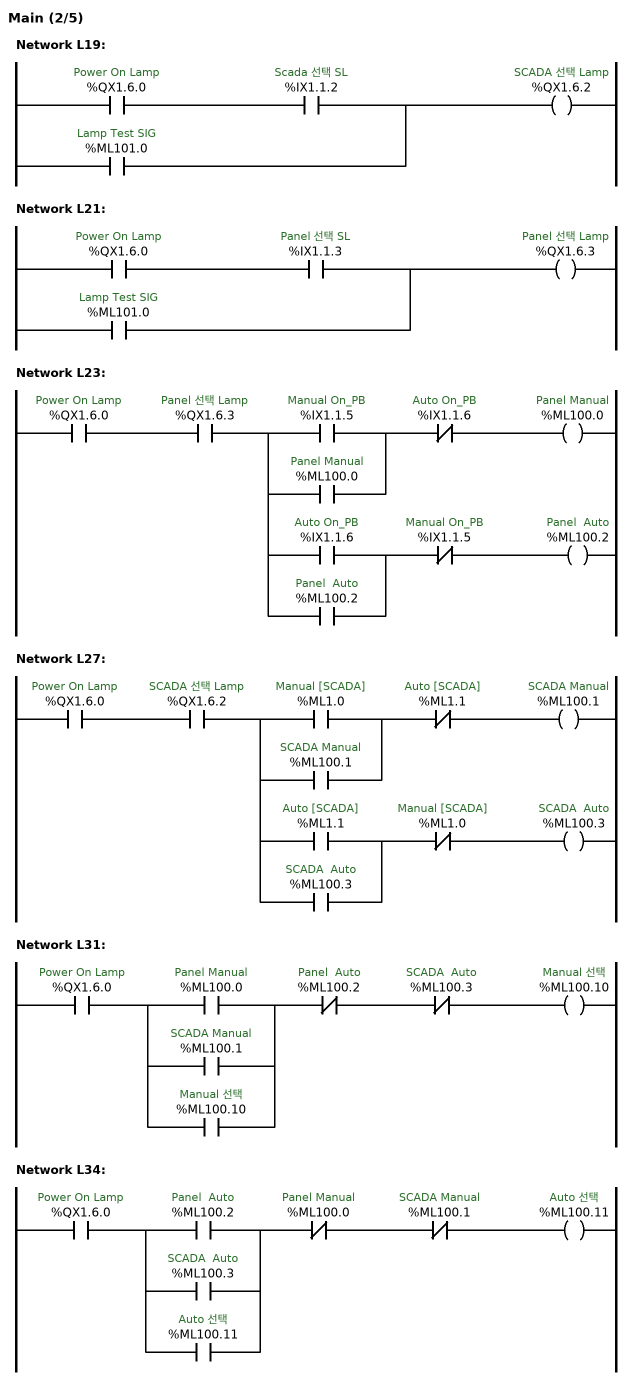
(* Rung L19 *)
%QX1.6.2 := (%QX1.6.0 AND %IX1.1.2) OR %ML101.0;
(* Rung L21 *)
%QX1.6.3 := (%QX1.6.0 AND %IX1.1.3) OR %ML101.0;
(* Rung L23 *)
%ML100.0 := %QX1.6.0 AND %QX1.6.3 AND (%IX1.1.5 OR %ML100.0) AND NOT %IX1.1.6;
%ML100.2 := %QX1.6.0 AND %QX1.6.3 AND (%IX1.1.6 OR %ML100.2) AND NOT %IX1.1.5;
(* Rung L27 *)
%ML100.1 := %QX1.6.0 AND %QX1.6.2 AND (%ML1.0 OR %ML100.1) AND NOT %ML1.1;
%ML100.3 := %QX1.6.0 AND %QX1.6.2 AND (%ML1.1 OR %ML100.3) AND NOT %ML1.0;
(* Rung L31 *)
%ML100.10 := %QX1.6.0 AND (%ML100.0 OR %ML100.1 OR %ML100.10) AND NOT %ML100.2 AND NOT %ML100.3;
(* Rung L34 *)
%ML100.11 := %QX1.6.0 AND (%ML100.2 OR %ML100.3 OR %ML100.11) AND NOT %ML100.0 AND NOT %ML100.1;

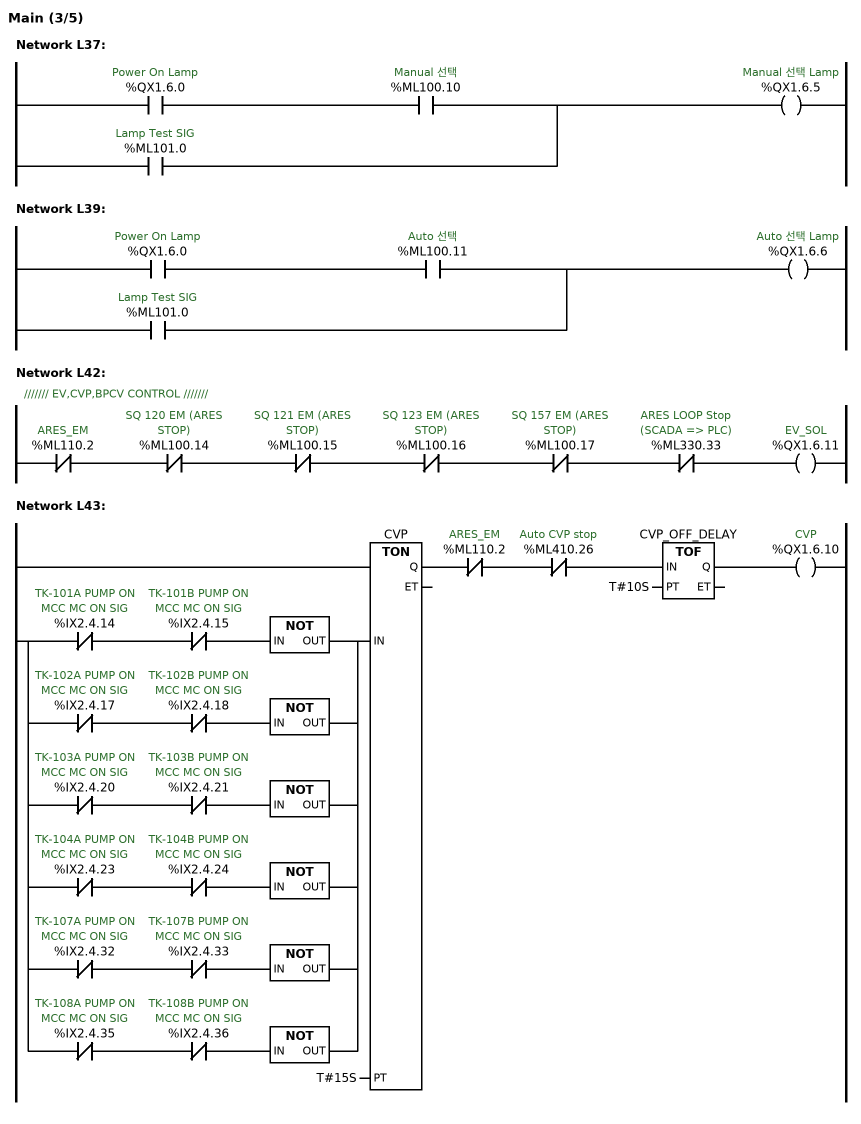
(* Rung L37 *)
%QX1.6.5 := (%QX1.6.0 AND %ML100.10) OR %ML101.0;
(* Rung L39 *)
%QX1.6.6 := (%QX1.6.0 AND %ML100.11) OR %ML101.0;
(* /////// EV,CVP,BPCV CONTROL /////// *)
(* Rung L42 *)
%QX1.6.11 := NOT %ML110.2 AND NOT %ML100.14 AND NOT %ML100.15 AND NOT %ML100.16 AND NOT %ML100.17 AND NOT %ML330.33;
(* Rung L43 *)
CVP(IN := (NOT (NOT %IX2.4.14 AND NOT %IX2.4.15)) OR (NOT (NOT %IX2.4.17 AND NOT %IX2.4.18)) OR (NOT (NOT %IX2.4.20 AND NOT %IX2.4.21)) OR (NOT (NOT %IX2.4.23 AND NOT %IX2.4.24)) OR (NOT (NOT %IX2.4.32 AND NOT %IX2.4.33)) OR (NOT (NOT %IX2.4.35 AND NOT %IX2.4.36)), PT := T#15S);
CVP_OFF_DELAY(IN := CVP.Q AND NOT %ML110.2 AND NOT %ML410.26, PT := T#10S);
%QX1.6.10 := CVP_OFF_DELAY.Q;

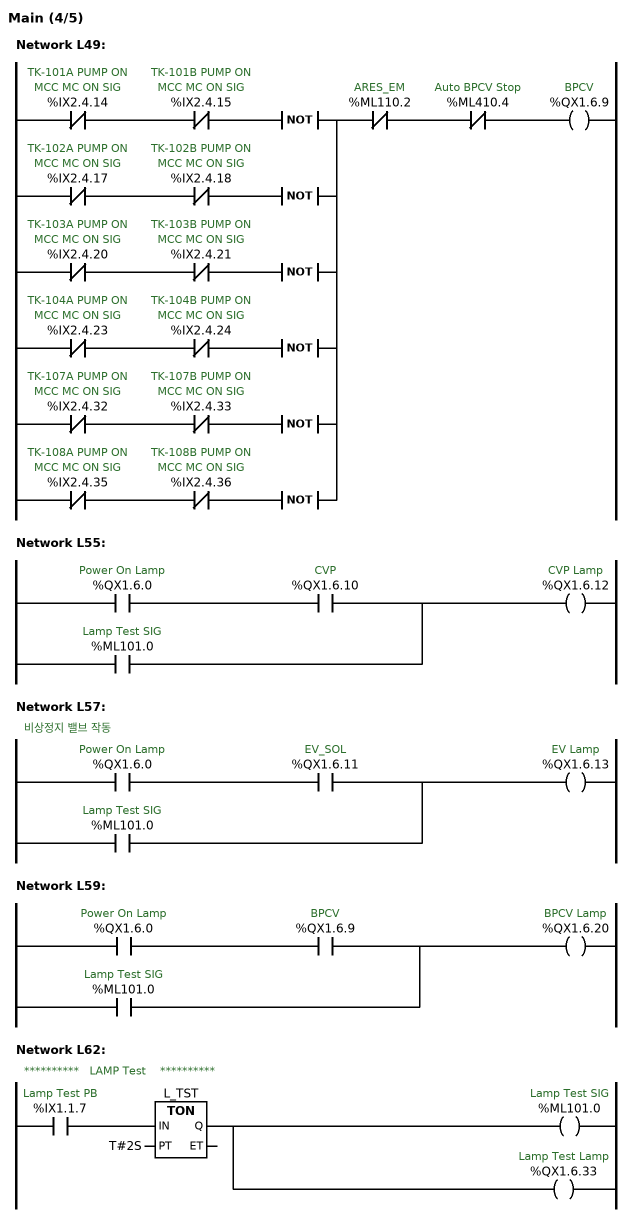
(* Rung L49 *)
%QX1.6.9 := (NOT (NOT %IX2.4.14 AND NOT %IX2.4.15) OR NOT (NOT %IX2.4.17 AND NOT %IX2.4.18) OR NOT (NOT %IX2.4.20 AND NOT %IX2.4.21) OR NOT (NOT %IX2.4.23 AND NOT %IX2.4.24) OR NOT (NOT %IX2.4.32 AND NOT %IX2.4.33) OR NOT (NOT %IX2.4.35 AND NOT %IX2.4.36)) AND NOT %ML110.2 AND NOT %ML410.4;
(* Rung L55 *)
%QX1.6.12 := (%QX1.6.0 AND %QX1.6.10) OR %ML101.0;
(* Rung L57 *)
%QX1.6.13 := (%QX1.6.0 AND %QX1.6.11) OR %ML101.0;
(* 비상정지 밸브 작동 *)
(* Rung L59 *)
%QX1.6.20 := (%QX1.6.0 AND %QX1.6.9) OR %ML101.0;
(* **********   LAMP Test    ********** *)
(* Rung L62 *)
L_TST(IN := %IX1.1.7, PT := T#2S);
%ML101.0 := L_TST.Q;
%QX1.6.33 := L_TST.Q;

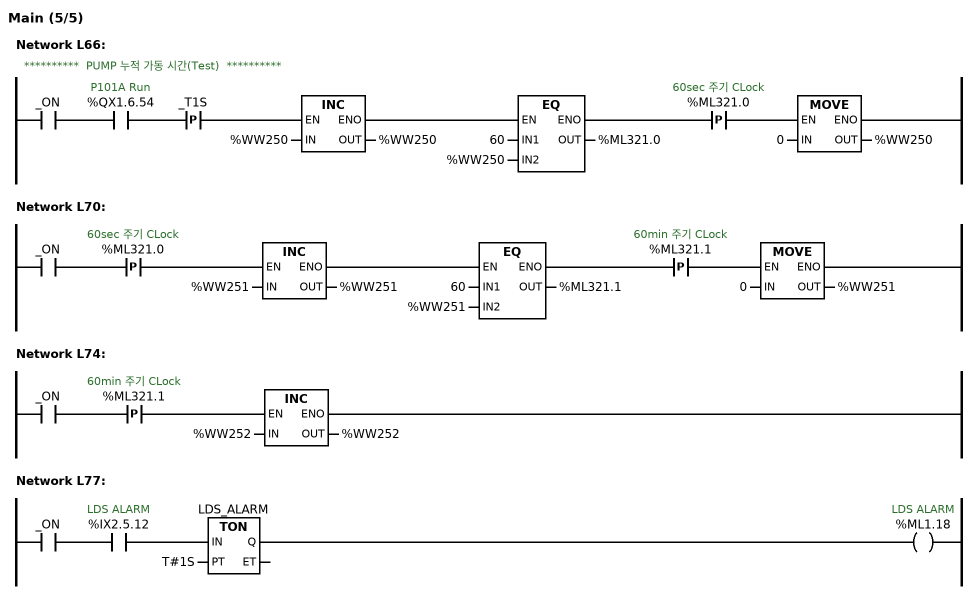
(* **********  PUMP 누적 가동 시간(Test)  ********** *)
(* Rung L66 *)
_e1(CLK := _T1S);
IF _ON AND %QX1.6.54 AND _e1.Q THEN
    %WW250 := INC(%WW250);
    %ML321.0 := 60 = %WW250;
END_IF;
_e2(CLK := %ML321.0);
IF _ON AND %QX1.6.54 AND _e1.Q AND _e2.Q THEN %WW250 := 0; END_IF;
(* Rung L70 *)
_e3(CLK := %ML321.0);
IF _ON AND _e3.Q THEN
    %WW251 := INC(%WW251);
    %ML321.1 := 60 = %WW251;
END_IF;
_e4(CLK := %ML321.1);
IF _ON AND _e3.Q AND _e4.Q THEN %WW251 := 0; END_IF;
(* Rung L74 *)
_e5(CLK := %ML321.1);
IF _ON AND _e5.Q THEN %WW252 := INC(%WW252); END_IF;
(* Rung L77 *)
LDS_ALARM(IN := _ON AND %IX2.5.12, PT := T#1S);
%ML1.18 := LDS_ALARM.Q;
END_PROGRAM

PROGRAM TK_LV_HH,LL_PumpStop (* task: 스캔 프로그램 *)

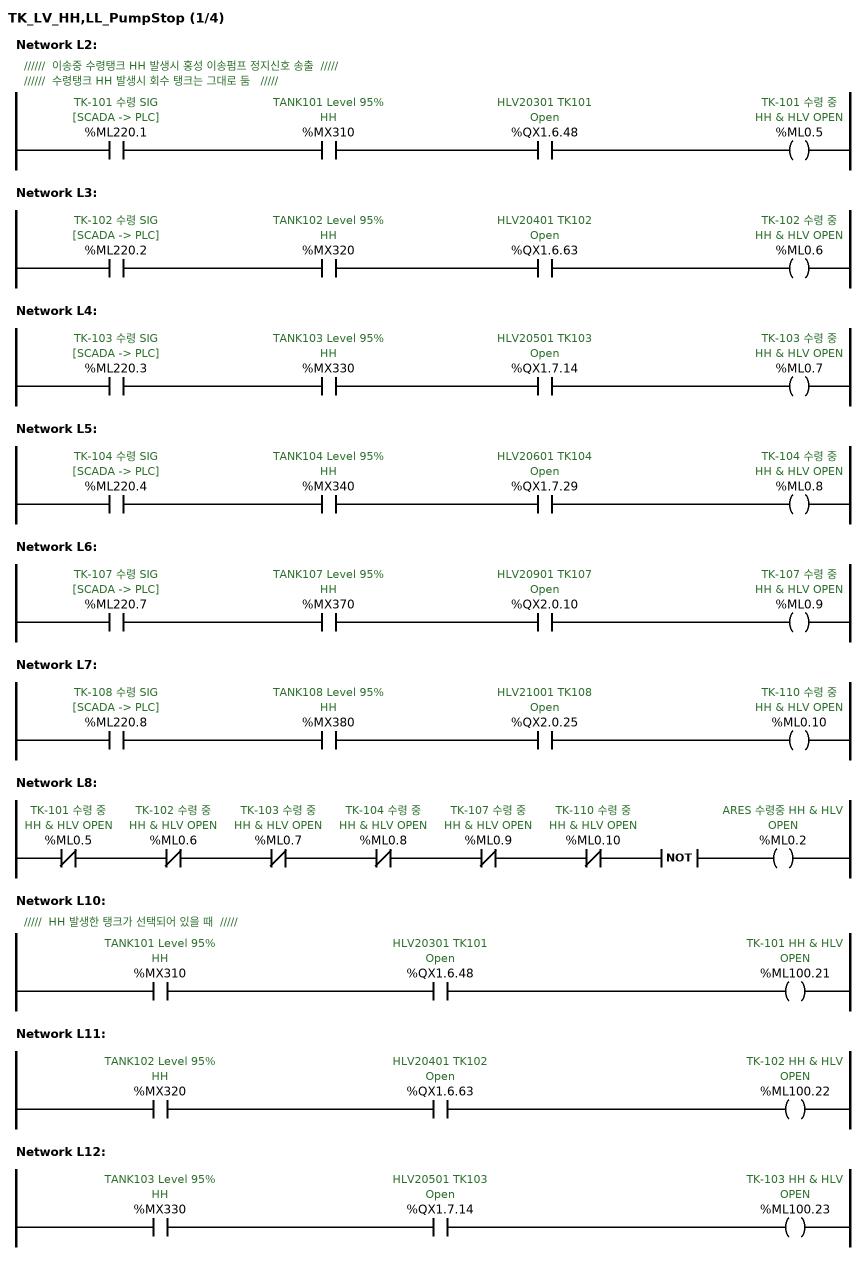
(* //////  이송중 수령탱크 HH 발생시 홍성 이송펌프 정지신호 송출  ///// *)
(* //////  수령탱크 HH 발생시 회수 탱크는 그대로 둠   ///// *)
(* Rung L2 *)
%ML0.5 := %ML220.1 AND %MX310 AND %QX1.6.48;
(* Rung L3 *)
%ML0.6 := %ML220.2 AND %MX320 AND %QX1.6.63;
(* Rung L4 *)
%ML0.7 := %ML220.3 AND %MX330 AND %QX1.7.14;
(* Rung L5 *)
%ML0.8 := %ML220.4 AND %MX340 AND %QX1.7.29;
(* Rung L6 *)
%ML0.9 := %ML220.7 AND %MX370 AND %QX2.0.10;
(* Rung L7 *)
%ML0.10 := %ML220.8 AND %MX380 AND %QX2.0.25;
(* Rung L8 *)
%ML0.2 := NOT (NOT %ML0.5 AND NOT %ML0.6 AND NOT %ML0.7 AND NOT %ML0.8 AND NOT %ML0.9 AND NOT %ML0.10);
(* /////  HH 발생한 탱크가 선택되어 있을 때  ///// *)
(* Rung L10 *)
%ML100.21 := %MX310 AND %QX1.6.48;
(* Rung L11 *)
%ML100.22 := %MX320 AND %QX1.6.63;
(* Rung L12 *)
%ML100.23 := %MX330 AND %QX1.7.14;

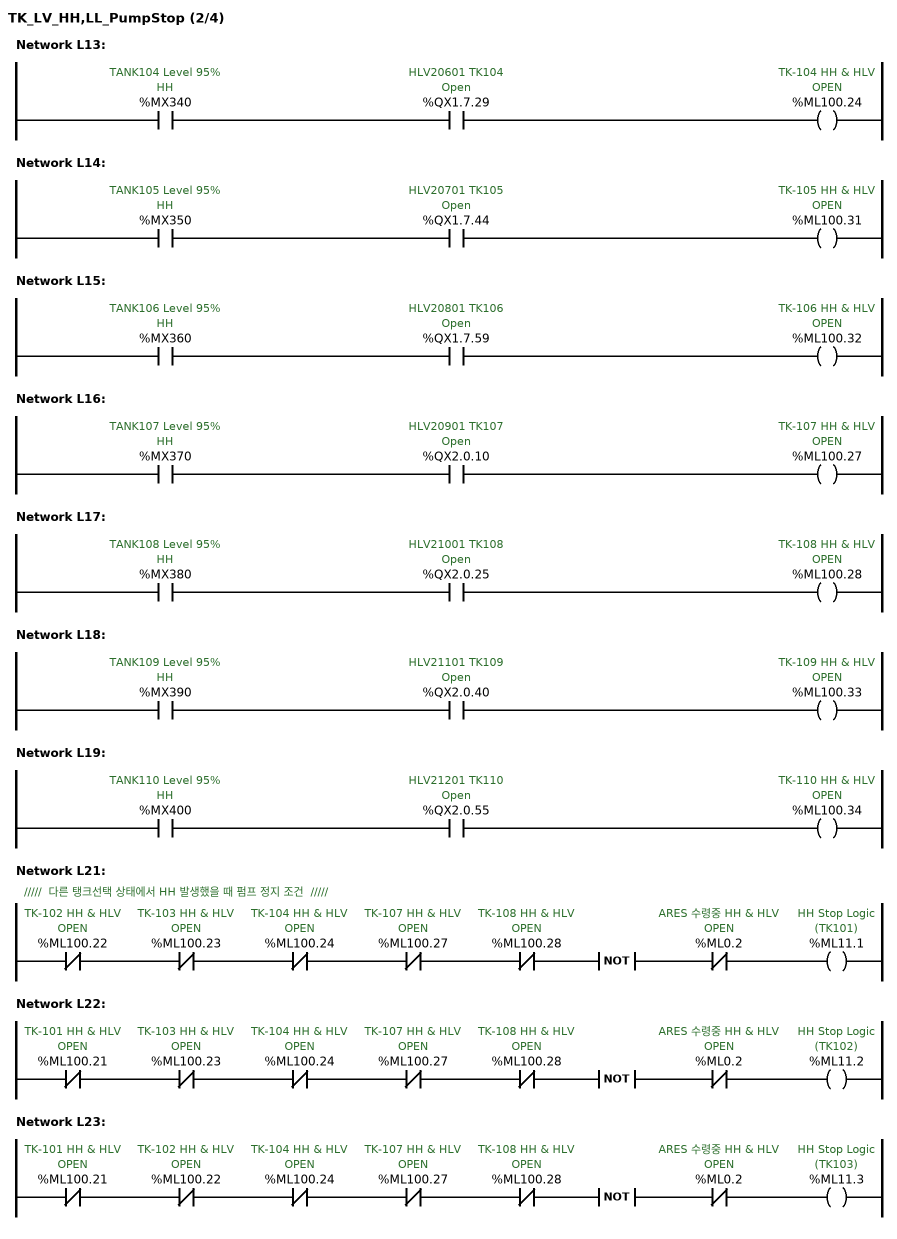
(* Rung L13 *)
%ML100.24 := %MX340 AND %QX1.7.29;
(* Rung L14 *)
%ML100.31 := %MX350 AND %QX1.7.44;
(* Rung L15 *)
%ML100.32 := %MX360 AND %QX1.7.59;
(* Rung L16 *)
%ML100.27 := %MX370 AND %QX2.0.10;
(* Rung L17 *)
%ML100.28 := %MX380 AND %QX2.0.25;
(* Rung L18 *)
%ML100.33 := %MX390 AND %QX2.0.40;
(* Rung L19 *)
%ML100.34 := %MX400 AND %QX2.0.55;
(* /////  다른 탱크선택 상태에서 HH 발생했을 때 펌프 정지 조건  ///// *)
(* Rung L21 *)
%ML11.1 := NOT (NOT %ML100.22 AND NOT %ML100.23 AND NOT %ML100.24 AND NOT %ML100.27 AND NOT %ML100.28) AND NOT %ML0.2;
(* Rung L22 *)
%ML11.2 := NOT (NOT %ML100.21 AND NOT %ML100.23 AND NOT %ML100.24 AND NOT %ML100.27 AND NOT %ML100.28) AND NOT %ML0.2;
(* Rung L23 *)
%ML11.3 := NOT (NOT %ML100.21 AND NOT %ML100.22 AND NOT %ML100.24 AND NOT %ML100.27 AND NOT %ML100.28) AND NOT %ML0.2;

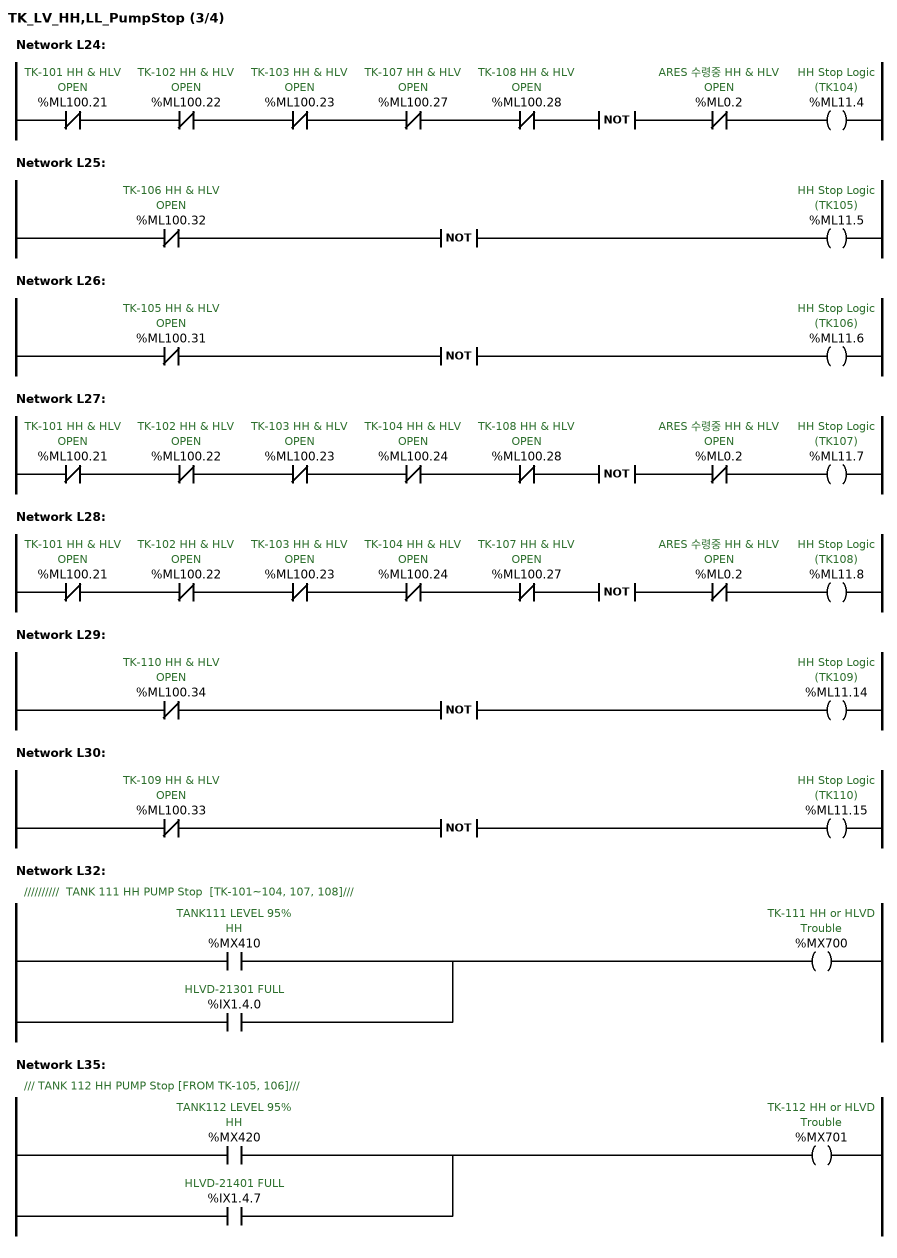
(* Rung L24 *)
%ML11.4 := NOT (NOT %ML100.21 AND NOT %ML100.22 AND NOT %ML100.23 AND NOT %ML100.27 AND NOT %ML100.28) AND NOT %ML0.2;
(* Rung L25 *)
%ML11.5 := %ML100.32;
(* Rung L26 *)
%ML11.6 := %ML100.31;
(* Rung L27 *)
%ML11.7 := NOT (NOT %ML100.21 AND NOT %ML100.22 AND NOT %ML100.23 AND NOT %ML100.24 AND NOT %ML100.28) AND NOT %ML0.2;
(* Rung L28 *)
%ML11.8 := NOT (NOT %ML100.21 AND NOT %ML100.22 AND NOT %ML100.23 AND NOT %ML100.24 AND NOT %ML100.27) AND NOT %ML0.2;
(* Rung L29 *)
%ML11.14 := %ML100.34;
(* Rung L30 *)
%ML11.15 := %ML100.33;
(* //////////  TANK 111 HH PUMP Stop  [TK-101~104, 107, 108]/// *)
(* Rung L32 *)
%MX700 := %MX410 OR %IX1.4.0;
(* /// TANK 112 HH PUMP Stop [FROM TK-105, 106]/// *)
(* Rung L35 *)
%MX701 := %MX420 OR %IX1.4.7;

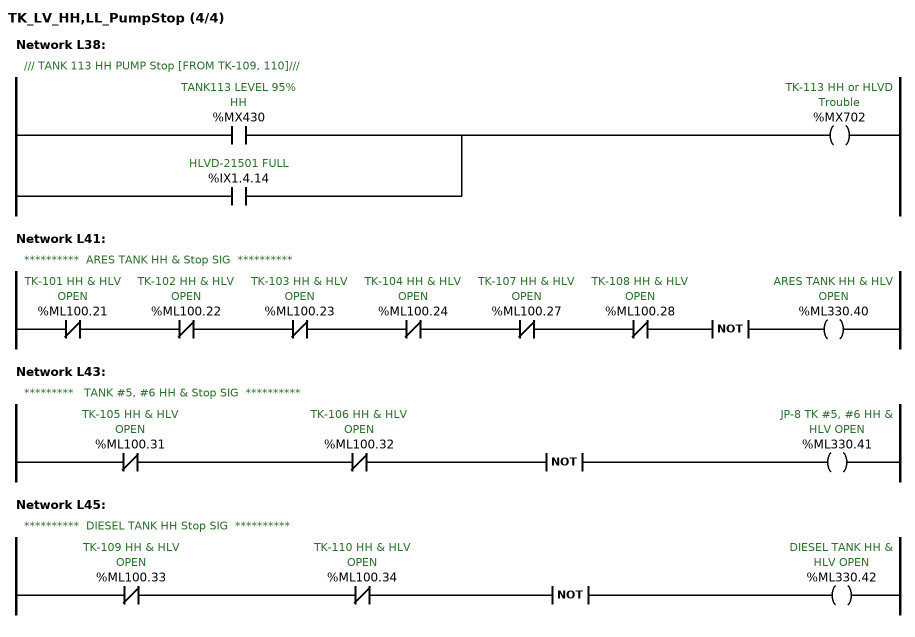
(* /// TANK 113 HH PUMP Stop [FROM TK-109, 110]/// *)
(* Rung L38 *)
%MX702 := %MX430 OR %IX1.4.14;
(* **********  ARES TANK HH & Stop SIG  ********** *)
(* Rung L41 *)
%ML330.40 := NOT (NOT %ML100.21 AND NOT %ML100.22 AND NOT %ML100.23 AND NOT %ML100.24 AND NOT %ML100.27 AND NOT %ML100.28);
(* *********   TANK #5, #6 HH & Stop SIG  ********** *)
(* Rung L43 *)
%ML330.41 := NOT (NOT %ML100.31 AND NOT %ML100.32);
(* **********  DIESEL TANK HH Stop SIG  ********** *)
(* Rung L45 *)
%ML330.42 := NOT (NOT %ML100.33 AND NOT %ML100.34);
END_PROGRAM

PROGRAM Automatic (* task: 스캔 프로그램 *)
VAR
    AHPC : TOF;
    AHPC1 : TOF;
    AHPC2 : TOF;
    ARES_LOOP_STOP : TOF; (* ARES_LOOP_Stop / SCADA => PLC *)
    ARES_LOOP_STOP1 : TOF; (* ARES_LOOP_Stop / SCADA => PLC *)
    ARES_LOOP_STOP2 : TON;
    ARES_LOOP_STOP3 : TON;
    ARES_LOOP_STOP4 : TON;
    AUTO_1ST_PUMP_STOP : TOF; (* 1차 펌프 정지 시 CVP우선 정지 후 펌프 지연 타이머 *)
    AUTO_1ST_PUMP_STOP1 : TON;
    AUTO_1ST_PUMP_STOP2 : TON;
    AUTO_1ST_PUMP_STOP3 : TON;
    AUTO_1ST_PUMP_STOP_CVP_HOLDING : TOF;
    Auto_restart_Alarm : TOF_RST;
    Auto_Restart_ea : FF;
    Auto_Restart_set : CTD_UINT;
    AUTO_SOCR : TON;
    Auto_Stating_ea : FF;
    AUTO_STR : TON;
    AUTO_STR1 : TON;
    AUTO_STR2 : TON;
    AUTO_S_FS : TON;
    INST : FF;
    INST1 : TOF;
    INST2 : TOF_RST;
    INST3 : TOF;
    INST4 : TOF;
    INST5 : TOF;
    INST6 : TON;
    j : TOF;
    L_TST : TON;
    one_set_run : TON;
    one_set_run1 : TON;
    one_set_run2 : TON;
    one_set_run3 : TON;
    one_set_run4 : TON;
    One_set_stp : TON;
    One_set_stp1 : TON;
    P110A_FS : TON;
    P110B_FS : TON;
    P110C_FS : TON;
    P111A_FS : TON;
    P112A_FS : TON;
    P1O10A_FS : TON;
    P1O10B_FS : TON;
    P1O10C_FS : TON;
    P1O11C_FS : TON;
    P1O12C_FS : TON;
    P1O13C_FS : TON;
    P1O18B_FS : TON;
    P1O6C_FS : TON;
    P1O7A_FS : TON;
    P1O7B_FS : TON;
    P1O7C_FS : TON;
    P1O8A_FS : TON;
    P1O8B_FS : TON;
    P1O8C_FS : TON;
    P1O9A_FS : TON;
    P1O9B_FS : TON;
    P1O9C_FS : TON;
    SQ_2ea_ON : BOOL; (* SQ_3ea_on *)
    TP21 : TP; (* P101A FS *)
    TP22 : TP; (* P101A FS *)
    TP23 : TP; (* P101A FS *)
    TP24 : TP; (* P101A FS *)
    TP25 : TP; (* P101A FS *)
    TP26 : TP; (* P101A FS *)
    TP27 : TP; (* P101A FS *)
    TP28 : TP; (* P101A FS *)
    TP29 : TP; (* P101A FS *)
    TP30 : TP; (* P101A FS *)
    TP31 : TP; (* P101A FS *)
    TP32 : TP; (* P101A FS *)
    Two_set_run : TON;
    Two_set_run1 : TON;
    Two_set_run2 : TON;
    Two_set_run3 : TON;
    Two_set_run4 : TON;
    Two_set_run5 : TON;
    Two_set_stp : TON;
    Two_set_stp1 : TON;
    Two_set_stp10 : TON;
    Two_set_stp11 : TON;
    Two_set_stp12 : TON;
    Two_set_stp13 : TON;
    Two_set_stp14 : TON;
    Two_set_stp15 : TON;
    Two_set_stp2 : TON;
    Two_set_stp3 : TON;
    Two_set_stp4 : TON;
    Two_set_stp5 : TON;
    Two_set_stp6 : TON;
    Two_set_stp7 : TON;
    Two_set_stp8 : TON;
    Two_set_stp9 : TON;
    _10n : BOOL;
END_VAR
VAR_EXTERNAL
    _0100_CH1_DATA : INT; (* AT %UW1.0.3 *) (* 아날로그입력 모듈: 채널1 변환값 *)
    _0100_CH3_DATA : INT; (* AT %UW1.0.5 *) (* 아날로그입력 모듈: 채널3 변환값 *)
    _Auto_re_count : BOOL;
END_VAR
VAR
    _t1 : BOOL;
    _t2 : DINT;
    _t3 : DINT;
END_VAR

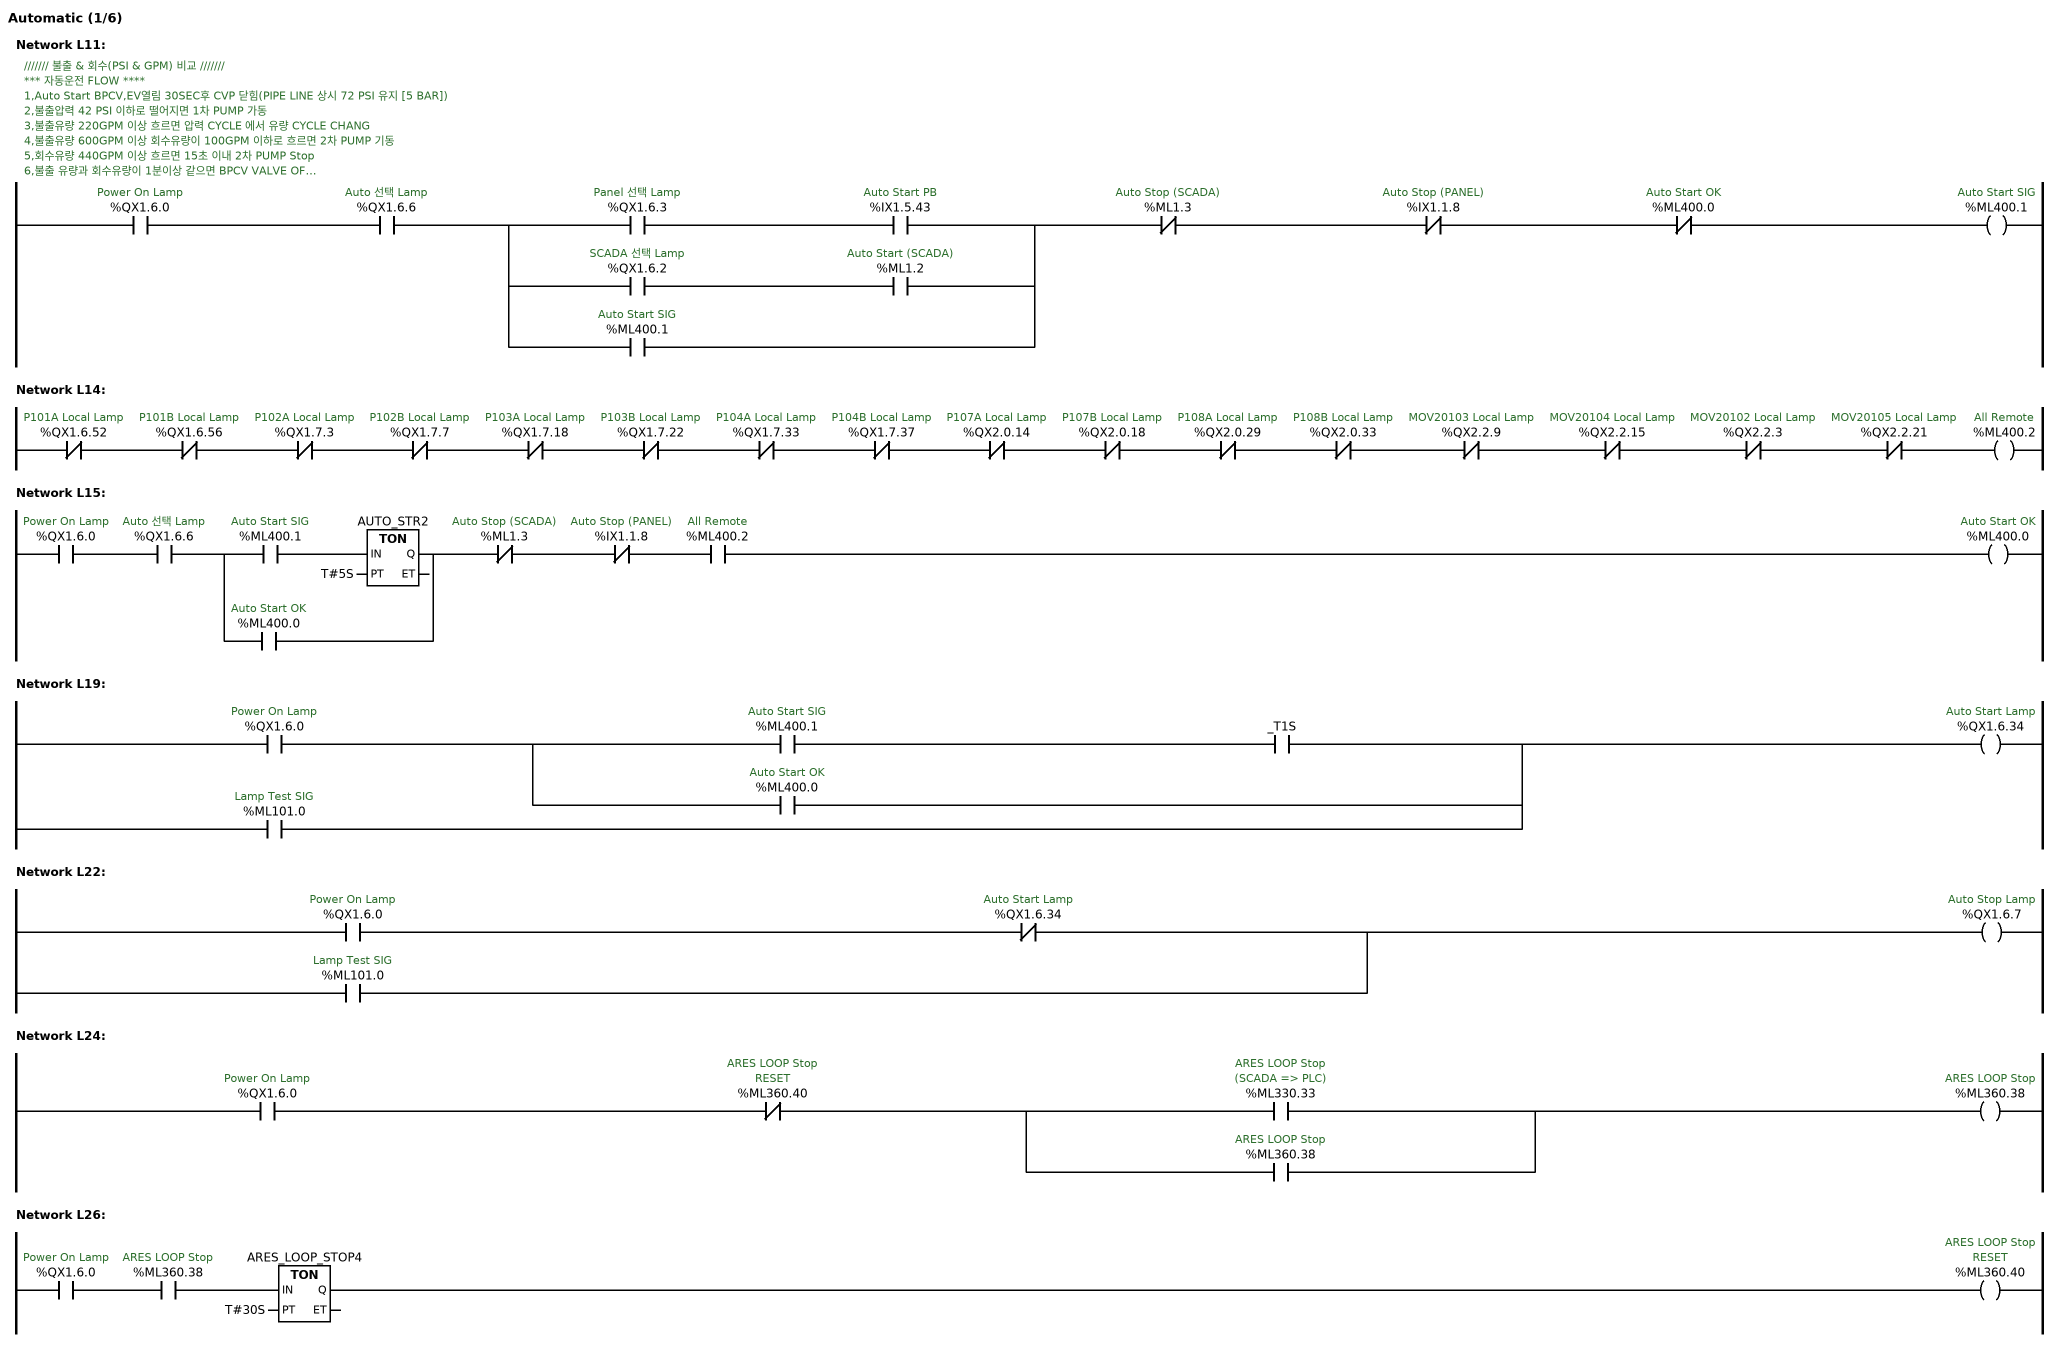
(* /////// 불출 & 회수(PSI & GPM) 비교 /////// *)
(* *** 자동운전 FLOW **** *)
(* 1,Auto Start BPCV,EV열림 30SEC후 CVP 닫힘(PIPE LINE 상시 72 PSI 유지 [5 BAR]) *)
(* 2,불출압력 42 PSI 이하로 떨어지면 1차 PUMP 가동 *)
(* 3,불출유량 220GPM 이상 흐르면 압력 CYCLE 에서 유량 CYCLE CHANG *)
(* 4,불출유량 600GPM 이상 회수유량이 100GPM 이하로 흐르면 2차 PUMP 기동 *)
(* 5,회수유량 440GPM 이상 흐르면 15초 이내 2차 PUMP Stop *)
(* 6,불출 유량과 회수유량이 1분이상 같으면 BPCV VALVE OFF *)
(* 7,불출 압력이 110PSI 1분이상 유지되면 1차PUMP Stop *)
(* *** TANK 7,8 번은 MOV OPEN 후 PUMP 기동 *** *)
(* /////// Auto RUNning READY /////// / (TK101,102,103,104,107,108 만 해당) *)
(* Rung L11 *)
%ML400.1 := %QX1.6.0 AND %QX1.6.6 AND ((%QX1.6.3 AND %IX1.5.43) OR (%QX1.6.2 AND %ML1.2) OR %ML400.1) AND NOT %ML1.3 AND NOT %IX1.1.8 AND NOT %ML400.0;
(* Rung L14 *)
%ML400.2 := NOT %QX1.6.52 AND NOT %QX1.6.56 AND NOT %QX1.7.3 AND NOT %QX1.7.7 AND NOT %QX1.7.18 AND NOT %QX1.7.22 AND NOT %QX1.7.33 AND NOT %QX1.7.37 AND NOT %QX2.0.14 AND NOT %QX2.0.18 AND NOT %QX2.0.29 AND NOT %QX2.0.33 AND NOT %QX2.2.9 AND NOT %QX2.2.15 AND NOT %QX2.2.3 AND NOT %QX2.2.21;
(* Rung L15 *)
AUTO_STR2(IN := %QX1.6.0 AND %QX1.6.6 AND %ML400.1, PT := T#5S);
%ML400.0 := (AUTO_STR2.Q OR (%QX1.6.0 AND %QX1.6.6 AND %ML400.0)) AND NOT %ML1.3 AND NOT %IX1.1.8 AND %ML400.2;
(* Rung L19 *)
%QX1.6.34 := (%QX1.6.0 AND ((%ML400.1 AND _T1S) OR %ML400.0)) OR %ML101.0;
(* Rung L22 *)
%QX1.6.7 := (%QX1.6.0 AND NOT %QX1.6.34) OR %ML101.0;
(* Rung L24 *)
%ML360.38 := %QX1.6.0 AND NOT %ML360.40 AND (%ML330.33 OR %ML360.38);
(* Rung L26 *)
ARES_LOOP_STOP4(IN := %QX1.6.0 AND %ML360.38, PT := T#30S);
%ML360.40 := ARES_LOOP_STOP4.Q;

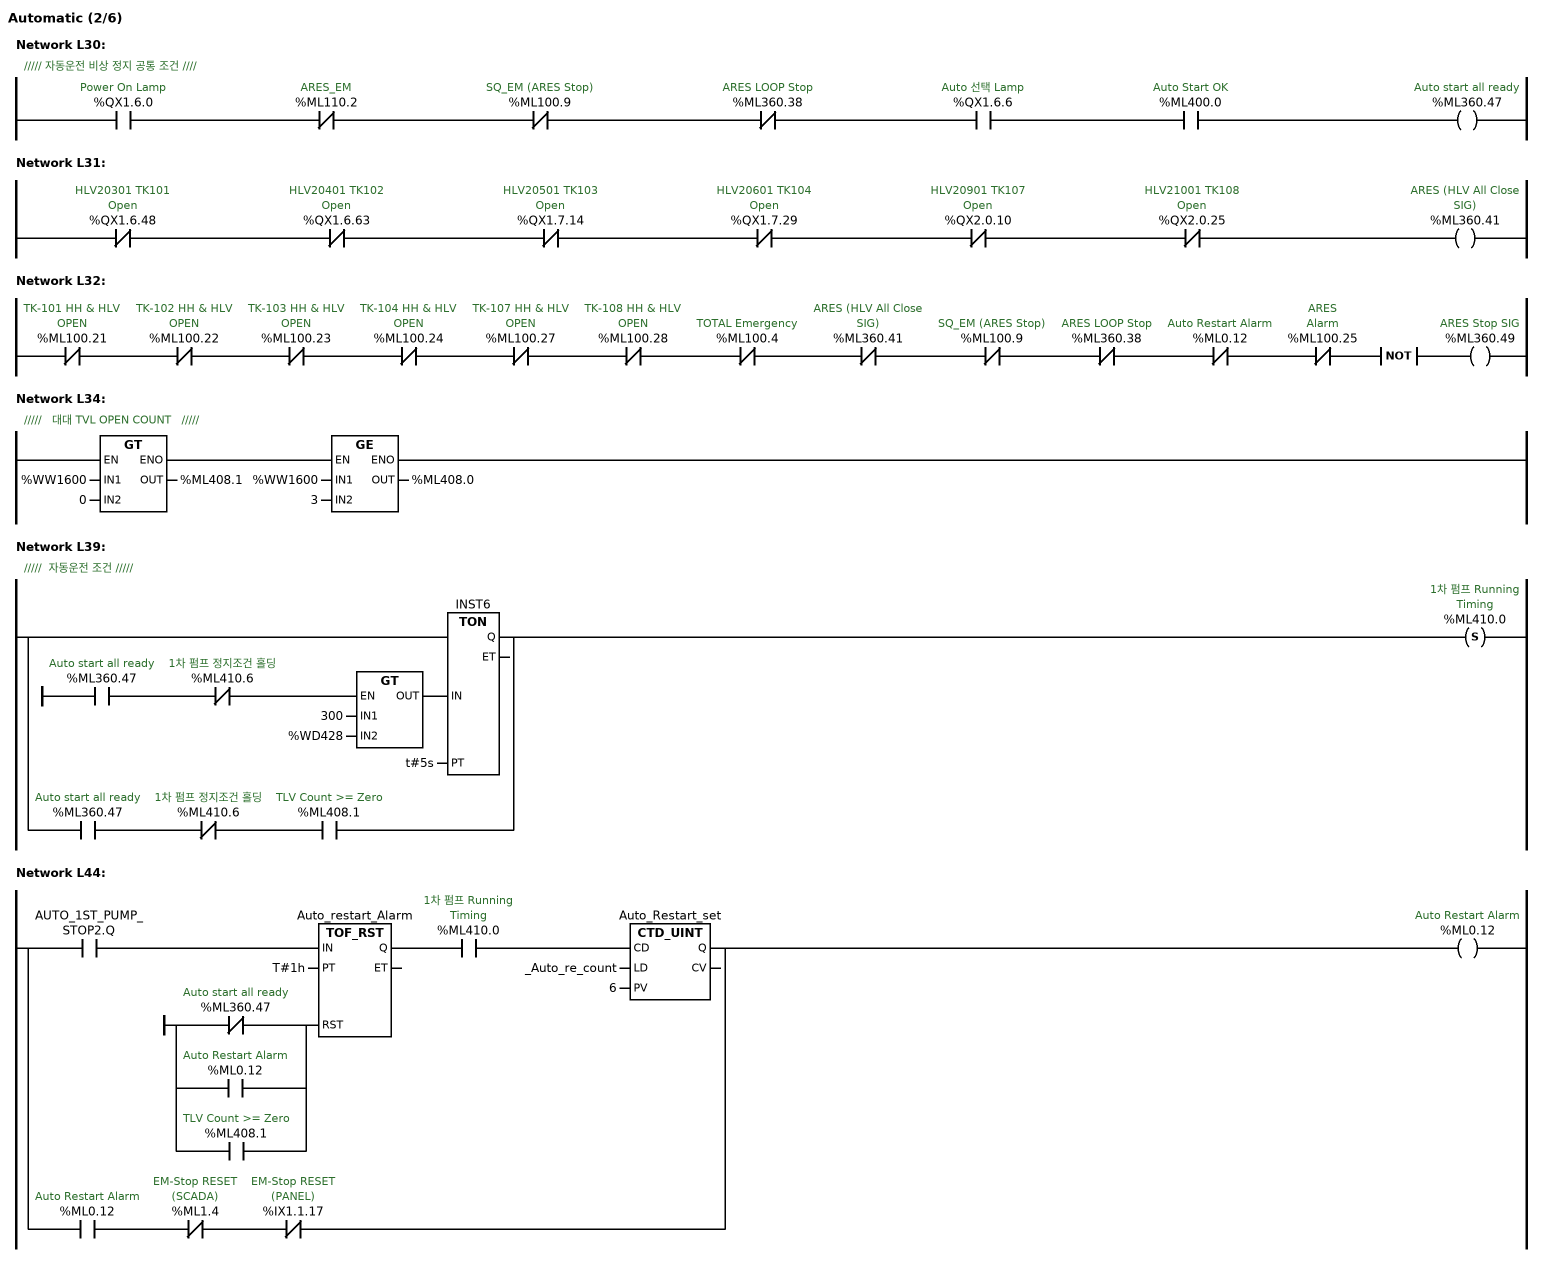
(* ///// 자동운전 비상 정지 공통 조건 //// *)
(* Rung L30 *)
%ML360.47 := %QX1.6.0 AND NOT %ML110.2 AND NOT %ML100.9 AND NOT %ML360.38 AND %QX1.6.6 AND %ML400.0;
(* Rung L31 *)
%ML360.41 := NOT %QX1.6.48 AND NOT %QX1.6.63 AND NOT %QX1.7.14 AND NOT %QX1.7.29 AND NOT %QX2.0.10 AND NOT %QX2.0.25;
(* Rung L32 *)
%ML360.49 := NOT (NOT %ML100.21 AND NOT %ML100.22 AND NOT %ML100.23 AND NOT %ML100.24 AND NOT %ML100.27 AND NOT %ML100.28 AND NOT %ML100.4 AND NOT %ML360.41 AND NOT %ML100.9 AND NOT %ML360.38 AND NOT %ML0.12 AND NOT %ML100.25);
(* /////   대대 TVL OPEN COUNT   ///// *)
(* Rung L34 *)
%ML408.1 := %WW1600 > 0;
%ML408.0 := %WW1600 >= 3;
(* /////  자동운전 조건 ///// *)
(* Rung L39 *)
IF %ML360.47 AND NOT %ML410.6 THEN _t1 := 300 > %WD428; END_IF;
INST6(IN := _t1, PT := t#5s);
IF INST6.Q OR (%ML360.47 AND NOT %ML410.6 AND %ML408.1) THEN %ML410.0 := TRUE; END_IF;
(* Rung L44 *)
Auto_restart_Alarm(IN := AUTO_1ST_PUMP_STOP2.Q, PT := T#1h, RST := NOT %ML360.47 OR %ML0.12 OR %ML408.1);
Auto_Restart_set(CD := Auto_restart_Alarm.Q AND %ML410.0, LD := _Auto_re_count, PV := 6);
%ML0.12 := Auto_Restart_set.Q OR (%ML0.12 AND NOT %ML1.4 AND NOT %IX1.1.17);

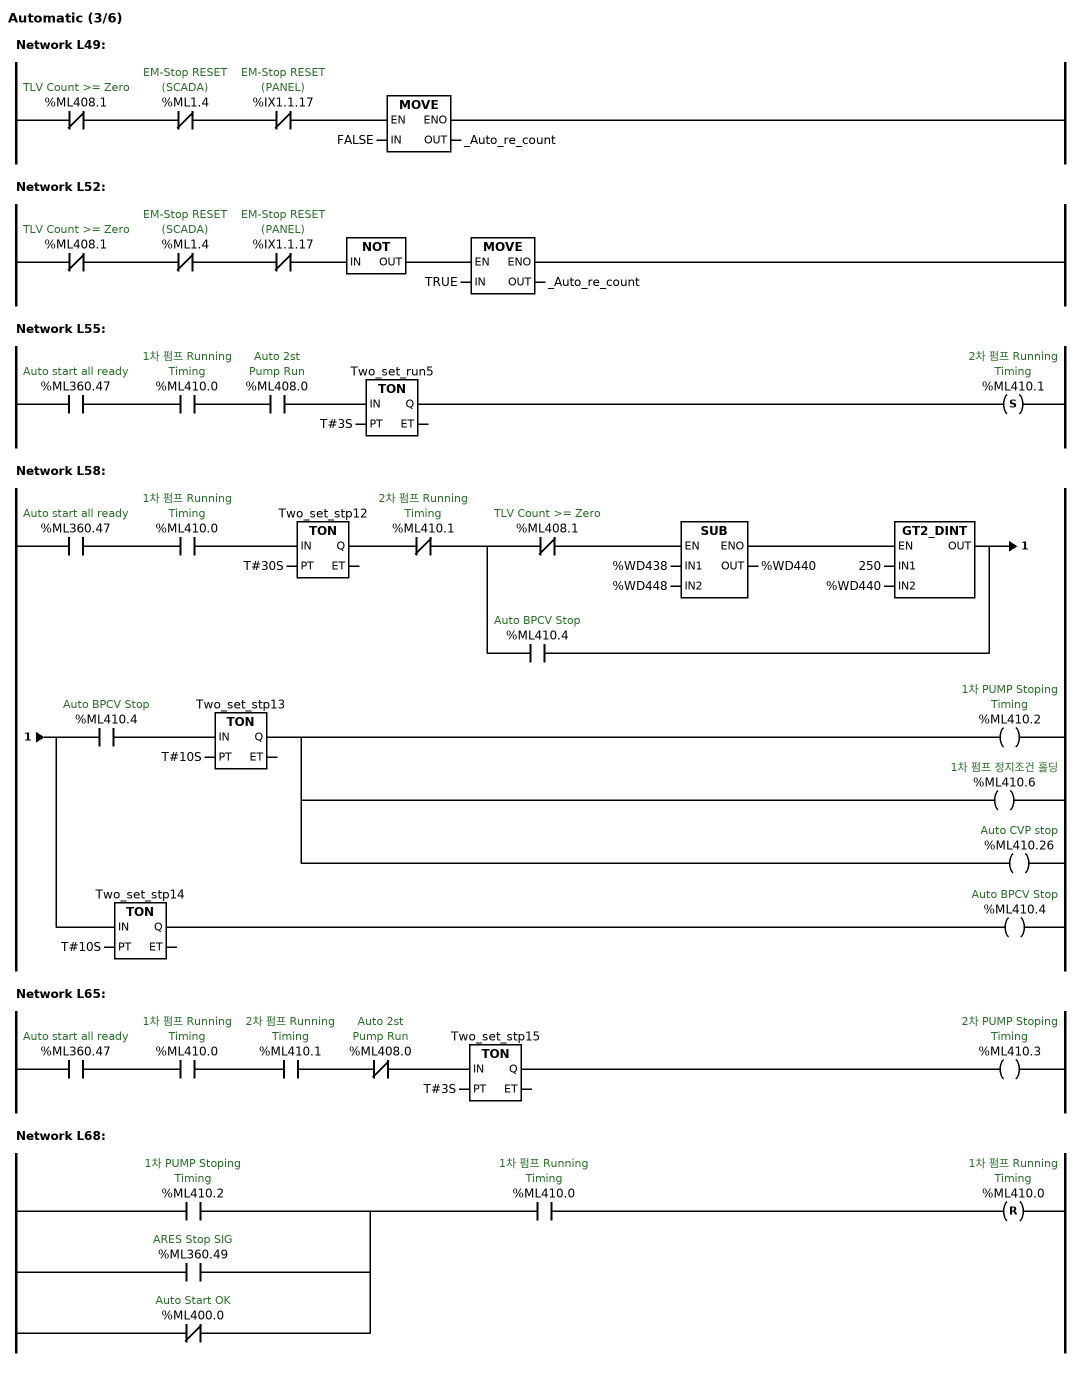
(* Rung L49 *)
IF NOT %ML408.1 AND NOT %ML1.4 AND NOT %IX1.1.17 THEN _Auto_re_count := FALSE; END_IF;
(* Rung L52 *)
IF NOT (NOT %ML408.1 AND NOT %ML1.4 AND NOT %IX1.1.17) THEN _Auto_re_count := TRUE; END_IF;
(* Rung L55 *)
Two_set_run5(IN := %ML360.47 AND %ML410.0 AND %ML408.0, PT := T#3S);
IF Two_set_run5.Q THEN %ML410.1 := TRUE; END_IF;
(* Rung L58 *)
Two_set_stp12(IN := %ML360.47 AND %ML410.0, PT := T#30S);
IF Two_set_stp12.Q AND NOT %ML410.1 AND NOT %ML408.1 THEN
    %WD440 := %WD438 - %WD448;
    _t2 := GT2_DINT(250, %WD440);
END_IF;
_t3 := _t2 OR (Two_set_stp12.Q AND NOT %ML410.1 AND %ML410.4);
Two_set_stp13(IN := _t3 AND %ML410.4, PT := T#10S);
%ML410.2 := Two_set_stp13.Q;
%ML410.6 := Two_set_stp13.Q;
%ML410.26 := Two_set_stp13.Q;
Two_set_stp14(IN := _t3, PT := T#10S);
%ML410.4 := Two_set_stp14.Q;
(* Rung L65 *)
Two_set_stp15(IN := %ML360.47 AND %ML410.0 AND %ML410.1 AND NOT %ML408.0, PT := T#3S);
%ML410.3 := Two_set_stp15.Q;
(* Rung L68 *)
IF (%ML410.2 OR %ML360.49 OR NOT %ML400.0) AND %ML410.0 THEN %ML410.0 := FALSE; END_IF;

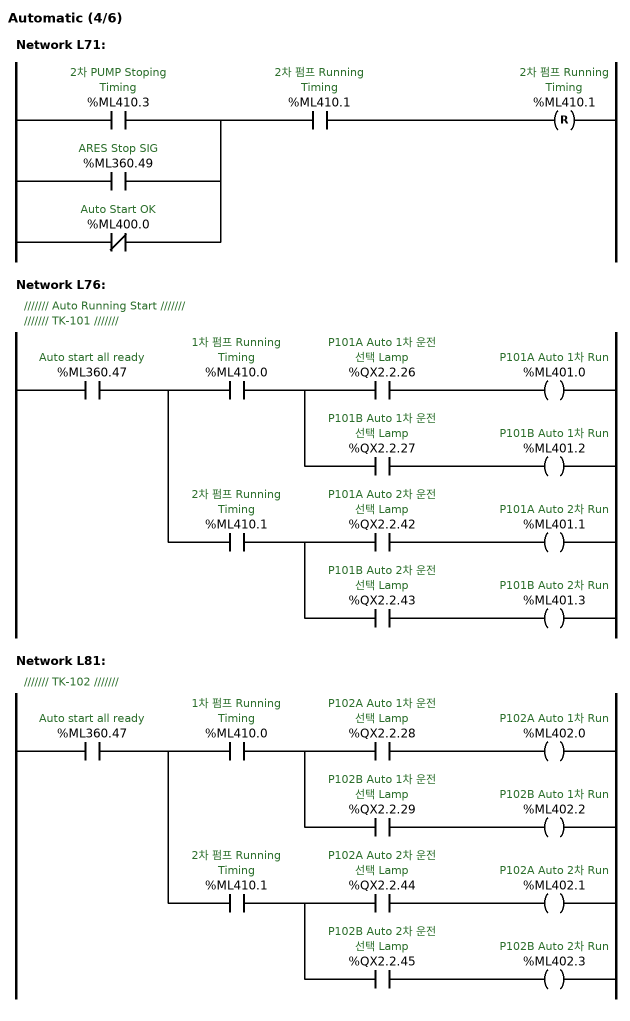
(* Rung L71 *)
IF (%ML410.3 OR %ML360.49 OR NOT %ML400.0) AND %ML410.1 THEN %ML410.1 := FALSE; END_IF;
(* /////// Auto Running Start /////// *)
(* /////// TK-101 /////// *)
(* Rung L76 *)
%ML401.0 := %ML360.47 AND %ML410.0 AND %QX2.2.26;
%ML401.2 := %ML360.47 AND %ML410.0 AND %QX2.2.27;
%ML401.1 := %ML360.47 AND %ML410.1 AND %QX2.2.42;
%ML401.3 := %ML360.47 AND %ML410.1 AND %QX2.2.43;
(* /////// TK-102 /////// *)
(* Rung L81 *)
%ML402.0 := %ML360.47 AND %ML410.0 AND %QX2.2.28;
%ML402.2 := %ML360.47 AND %ML410.0 AND %QX2.2.29;
%ML402.1 := %ML360.47 AND %ML410.1 AND %QX2.2.44;
%ML402.3 := %ML360.47 AND %ML410.1 AND %QX2.2.45;

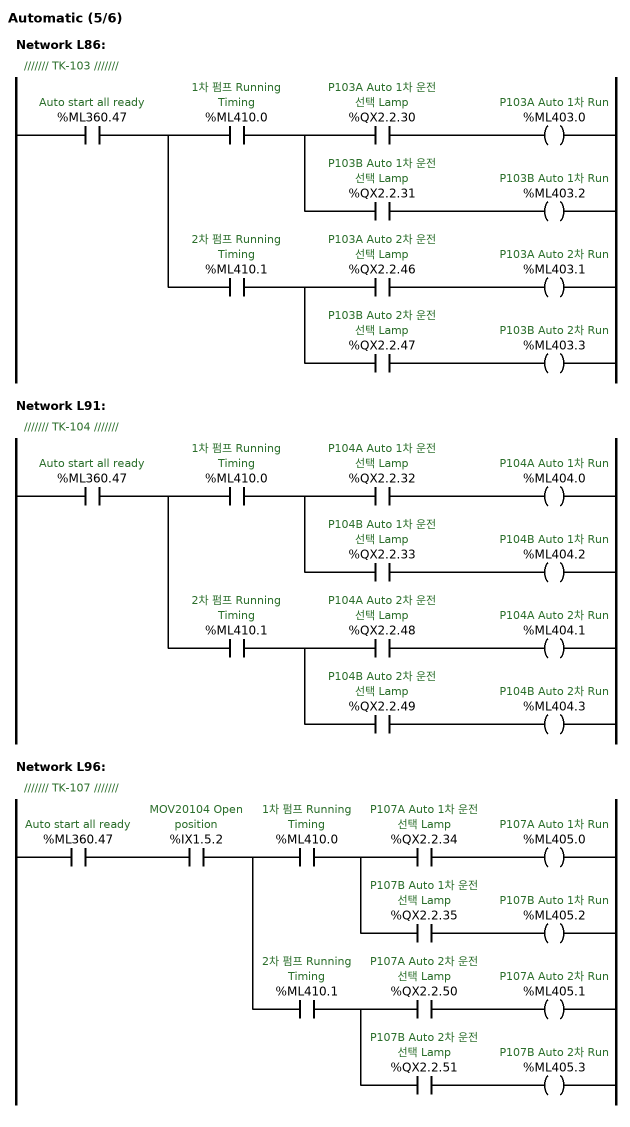
(* /////// TK-103 /////// *)
(* Rung L86 *)
%ML403.0 := %ML360.47 AND %ML410.0 AND %QX2.2.30;
%ML403.2 := %ML360.47 AND %ML410.0 AND %QX2.2.31;
%ML403.1 := %ML360.47 AND %ML410.1 AND %QX2.2.46;
%ML403.3 := %ML360.47 AND %ML410.1 AND %QX2.2.47;
(* /////// TK-104 /////// *)
(* Rung L91 *)
%ML404.0 := %ML360.47 AND %ML410.0 AND %QX2.2.32;
%ML404.2 := %ML360.47 AND %ML410.0 AND %QX2.2.33;
%ML404.1 := %ML360.47 AND %ML410.1 AND %QX2.2.48;
%ML404.3 := %ML360.47 AND %ML410.1 AND %QX2.2.49;
(* /////// TK-107 /////// *)
(* Rung L96 *)
%ML405.0 := %ML360.47 AND %IX1.5.2 AND %ML410.0 AND %QX2.2.34;
%ML405.2 := %ML360.47 AND %IX1.5.2 AND %ML410.0 AND %QX2.2.35;
%ML405.1 := %ML360.47 AND %IX1.5.2 AND %ML410.1 AND %QX2.2.50;
%ML405.3 := %ML360.47 AND %IX1.5.2 AND %ML410.1 AND %QX2.2.51;

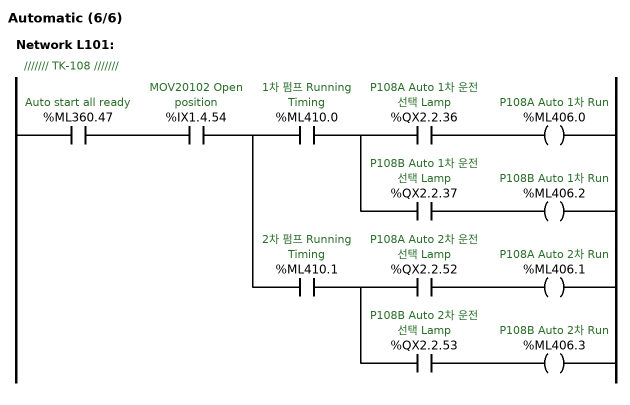
(* /////// TK-108 /////// *)
(* Rung L101 *)
%ML406.0 := %ML360.47 AND %IX1.4.54 AND %ML410.0 AND %QX2.2.36;
%ML406.2 := %ML360.47 AND %IX1.4.54 AND %ML410.0 AND %QX2.2.37;
%ML406.1 := %ML360.47 AND %IX1.4.54 AND %ML410.1 AND %QX2.2.52;
%ML406.3 := %ML360.47 AND %IX1.4.54 AND %ML410.1 AND %QX2.2.53;
END_PROGRAM

PROGRAM Manual_Tank_1,2,3,4,7,8 (* task: 스캔 프로그램 *)
VAR
    INST : ARY_GETE_DWORD;
    P101A_FS : TON; (* P101A_FS Alarm TON *)
    P101B_FS : TON;
    P101C_FS : TON;
    P102A_FS : TON;
    P102B_FS : TON;
    P102C_FS : TON;
    P103A_FS : TON;
    P103B_FS : TON;
    P103C_FS : TON;
    P104A_FS : TON;
    P104B_FS : TON;
    P104C_FS : TON;
    P105A_FS : TON; (* P101A_FS Alarm TON *)
    P105B_FS : TON;
    P105C_FS : TON;
    P106A_FS : TON;
    P106B_FS : TON;
    P106C_FS : TON;
    P107A_FS : TON;
    P107B_FS : TON;
    P107C_FS : TON;
    P108A_FS : TON;
    P108B_FS : TON;
    P108C_FS : TON;
    P109A_FS : TON;
    P109B_FS : TON;
    P109C_FS : TON;
    P110A_FS : TON;
    P110B_FS : TON;
    P110C_FS : TON;
    P111A_FS : TON;
    P111B_FS : TON;
    P111C_FS : TON;
    P112A_FS : TON;
    P112B_FS : TON;
    P112C_FS : TON;
END_VAR

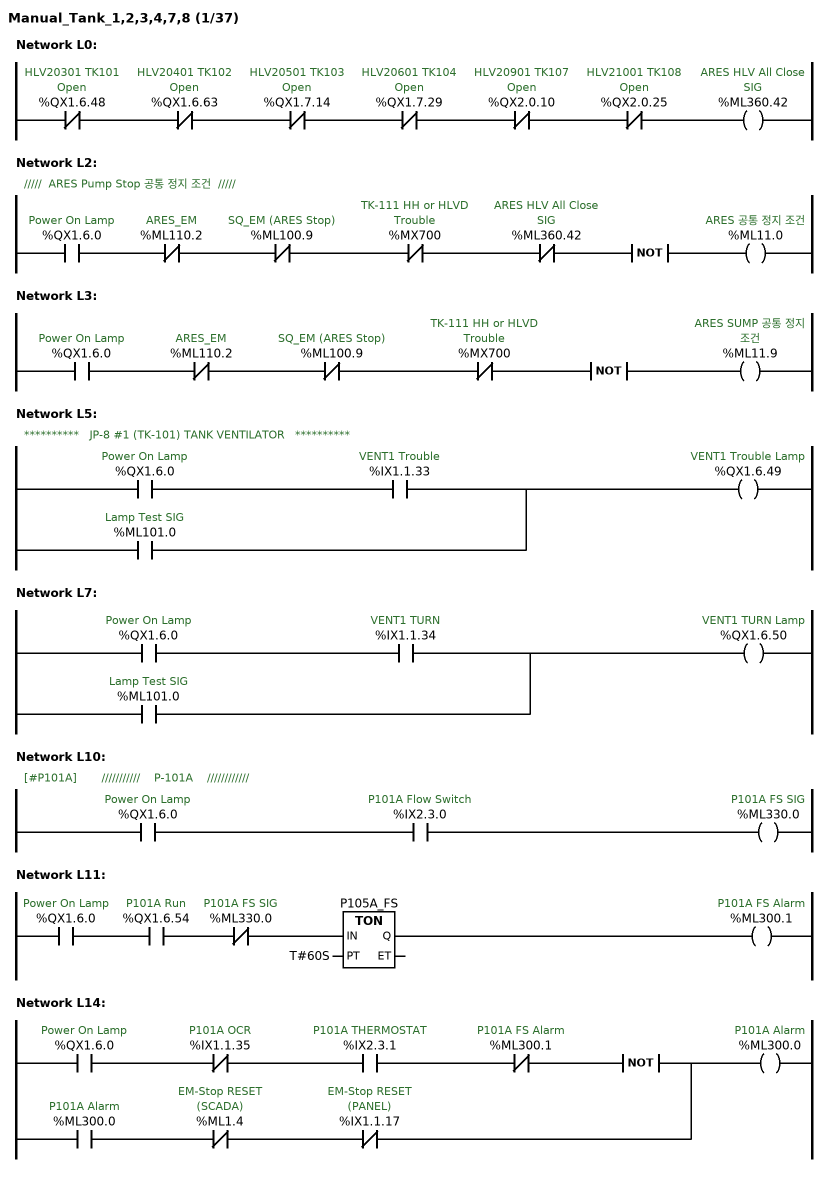
(* Rung L0 *)
%ML360.42 := NOT %QX1.6.48 AND NOT %QX1.6.63 AND NOT %QX1.7.14 AND NOT %QX1.7.29 AND NOT %QX2.0.10 AND NOT %QX2.0.25;
(* /////  ARES Pump Stop 공통 정지 조건  ///// *)
(* Rung L2 *)
%ML11.0 := NOT (%QX1.6.0 AND NOT %ML110.2 AND NOT %ML100.9 AND NOT %MX700 AND NOT %ML360.42);
(* Rung L3 *)
%ML11.9 := NOT (%QX1.6.0 AND NOT %ML110.2 AND NOT %ML100.9 AND NOT %MX700);
(* **********   JP-8 #1 (TK-101) TANK VENTILATOR   ********** *)
(* Rung L5 *)
%QX1.6.49 := (%QX1.6.0 AND %IX1.1.33) OR %ML101.0;
(* Rung L7 *)
%QX1.6.50 := (%QX1.6.0 AND %IX1.1.34) OR %ML101.0;
(* [#P101A]       ///////////    P-101A    //////////// *)
(* Rung L10 *)
%ML330.0 := %QX1.6.0 AND %IX2.3.0;
(* Rung L11 *)
P105A_FS(IN := %QX1.6.0 AND %QX1.6.54 AND NOT %ML330.0, PT := T#60S);
%ML300.1 := P105A_FS.Q;
(* Rung L14 *)
%ML300.0 := NOT (%QX1.6.0 AND NOT %IX1.1.35 AND %IX2.3.1 AND NOT %ML300.1) OR (%ML300.0 AND NOT %ML1.4 AND NOT %IX1.1.17);

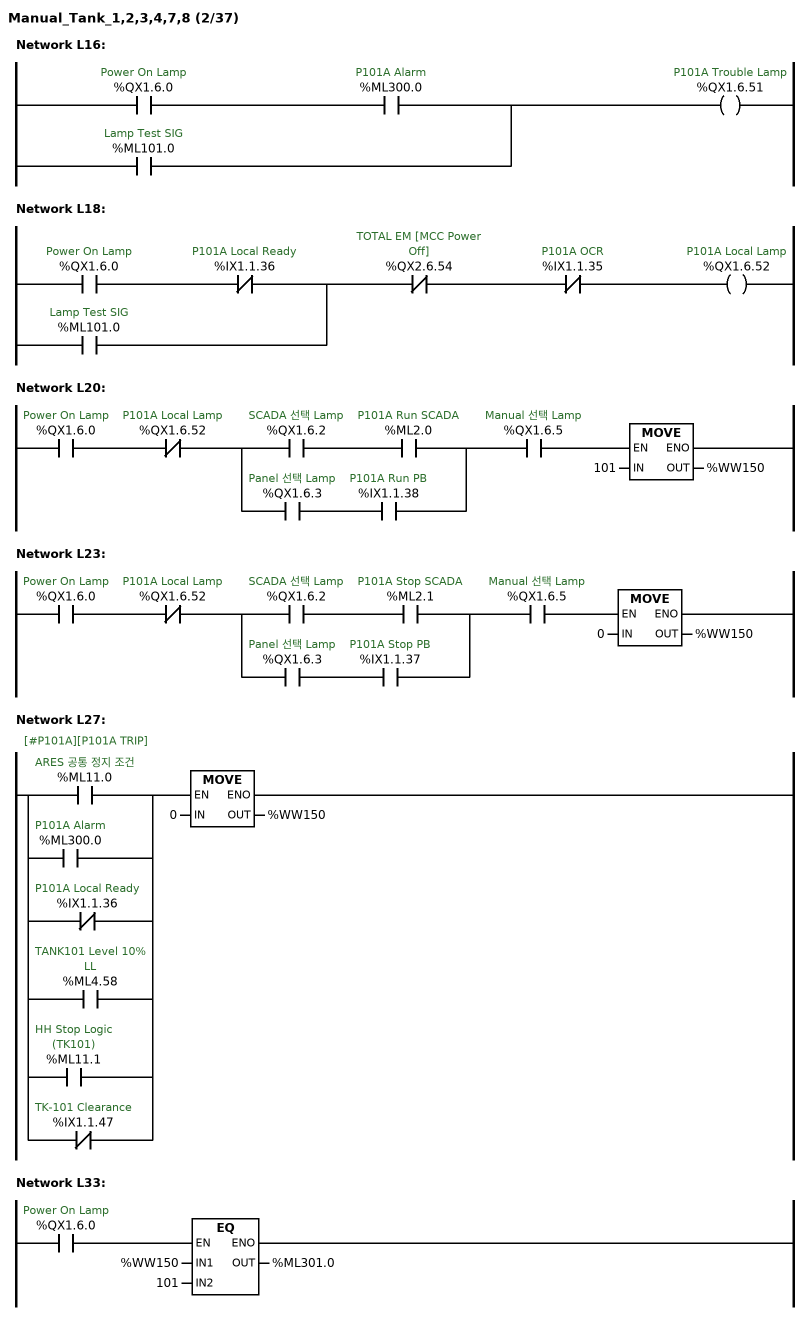
(* Rung L16 *)
%QX1.6.51 := (%QX1.6.0 AND %ML300.0) OR %ML101.0;
(* Rung L18 *)
%QX1.6.52 := ((%QX1.6.0 AND NOT %IX1.1.36) OR %ML101.0) AND NOT %QX2.6.54 AND NOT %IX1.1.35;
(* Rung L20 *)
IF %QX1.6.0 AND NOT %QX1.6.52 AND ((%QX1.6.2 AND %ML2.0) OR (%QX1.6.3 AND %IX1.1.38)) AND %QX1.6.5 THEN
    %WW150 := 101;
END_IF;
(* Rung L23 *)
IF %QX1.6.0 AND NOT %QX1.6.52 AND ((%QX1.6.2 AND %ML2.1) OR (%QX1.6.3 AND %IX1.1.37)) AND %QX1.6.5 THEN
    %WW150 := 0;
END_IF;
(* [#P101A][P101A TRIP] *)
(* Rung L27 *)
IF %ML11.0 OR %ML300.0 OR NOT %IX1.1.36 OR %ML4.58 OR %ML11.1 OR NOT %IX1.1.47 THEN %WW150 := 0; END_IF;
(* Rung L33 *)
IF %QX1.6.0 THEN %ML301.0 := %WW150 = 101; END_IF;

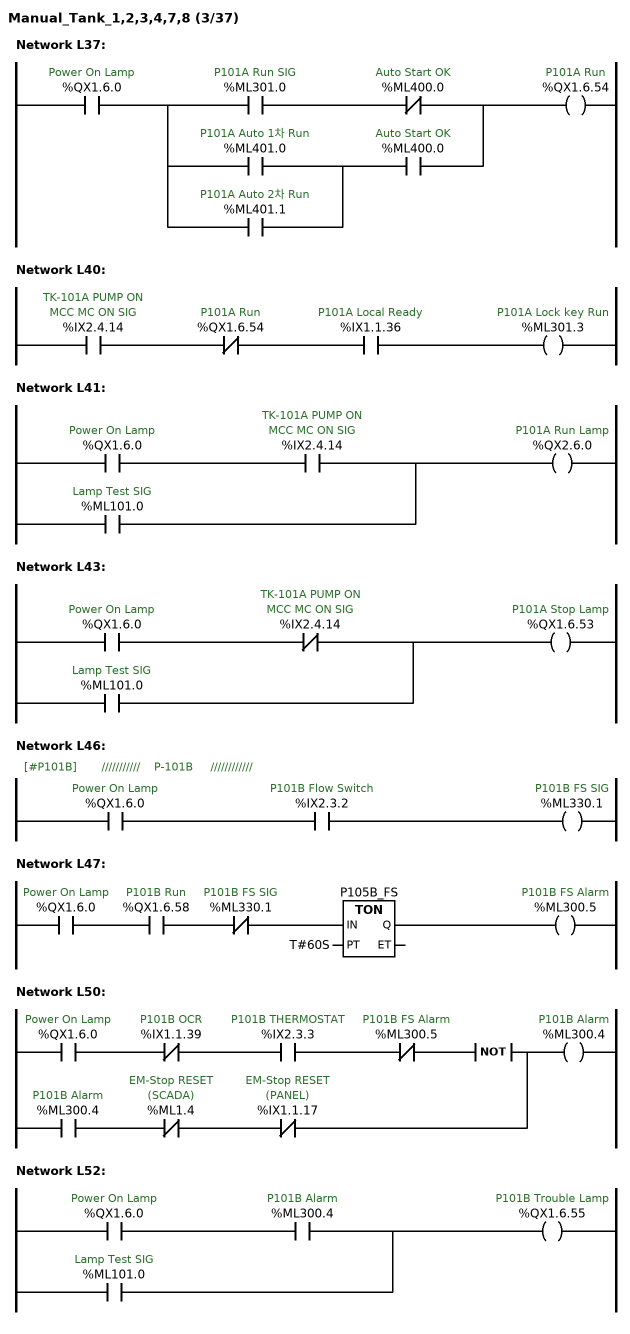
(* Rung L37 *)
%QX1.6.54 := %QX1.6.0 AND ((%ML301.0 AND NOT %ML400.0) OR ((%ML401.0 OR %ML401.1) AND %ML400.0));
(* Rung L40 *)
%ML301.3 := %IX2.4.14 AND NOT %QX1.6.54 AND %IX1.1.36;
(* Rung L41 *)
%QX2.6.0 := (%QX1.6.0 AND %IX2.4.14) OR %ML101.0;
(* Rung L43 *)
%QX1.6.53 := (%QX1.6.0 AND NOT %IX2.4.14) OR %ML101.0;
(* [#P101B]       ///////////    P-101B     //////////// *)
(* Rung L46 *)
%ML330.1 := %QX1.6.0 AND %IX2.3.2;
(* Rung L47 *)
P105B_FS(IN := %QX1.6.0 AND %QX1.6.58 AND NOT %ML330.1, PT := T#60S);
%ML300.5 := P105B_FS.Q;
(* Rung L50 *)
%ML300.4 := NOT (%QX1.6.0 AND NOT %IX1.1.39 AND %IX2.3.3 AND NOT %ML300.5) OR (%ML300.4 AND NOT %ML1.4 AND NOT %IX1.1.17);
(* Rung L52 *)
%QX1.6.55 := (%QX1.6.0 AND %ML300.4) OR %ML101.0;

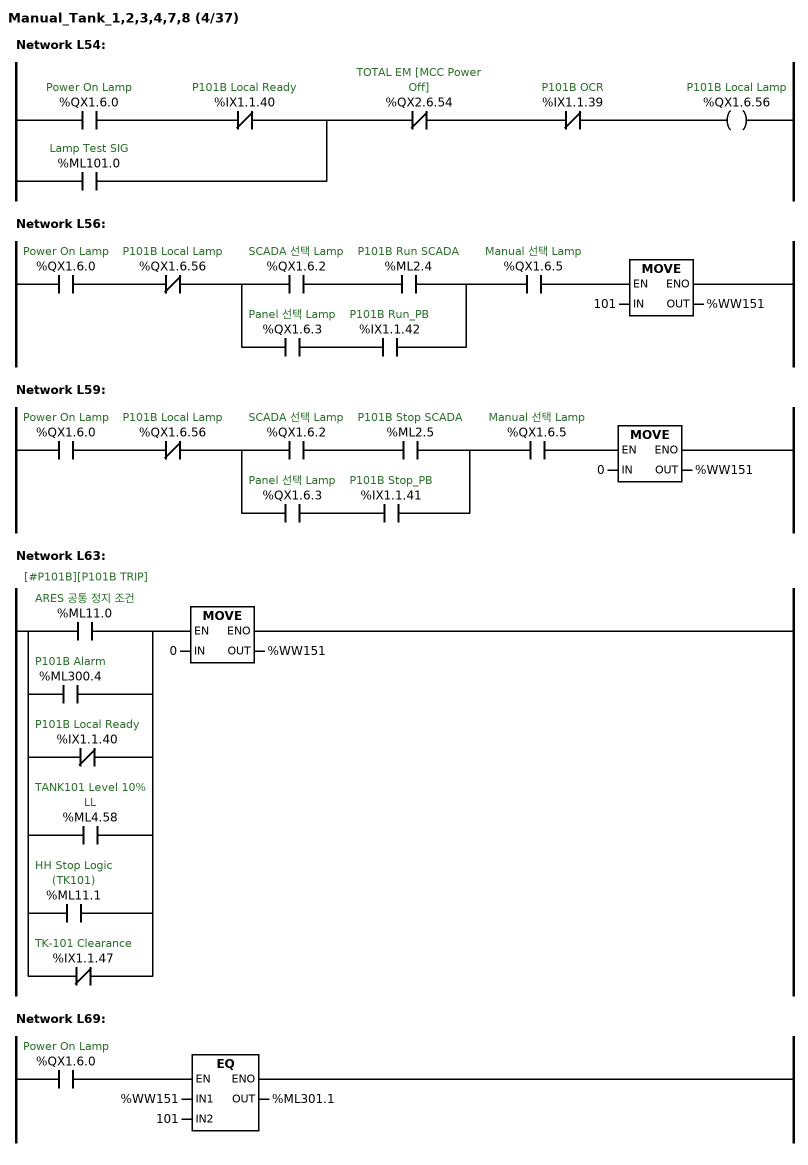
(* Rung L54 *)
%QX1.6.56 := ((%QX1.6.0 AND NOT %IX1.1.40) OR %ML101.0) AND NOT %QX2.6.54 AND NOT %IX1.1.39;
(* Rung L56 *)
IF %QX1.6.0 AND NOT %QX1.6.56 AND ((%QX1.6.2 AND %ML2.4) OR (%QX1.6.3 AND %IX1.1.42)) AND %QX1.6.5 THEN
    %WW151 := 101;
END_IF;
(* Rung L59 *)
IF %QX1.6.0 AND NOT %QX1.6.56 AND ((%QX1.6.2 AND %ML2.5) OR (%QX1.6.3 AND %IX1.1.41)) AND %QX1.6.5 THEN
    %WW151 := 0;
END_IF;
(* [#P101B][P101B TRIP] *)
(* Rung L63 *)
IF %ML11.0 OR %ML300.4 OR NOT %IX1.1.40 OR %ML4.58 OR %ML11.1 OR NOT %IX1.1.47 THEN %WW151 := 0; END_IF;
(* Rung L69 *)
IF %QX1.6.0 THEN %ML301.1 := %WW151 = 101; END_IF;

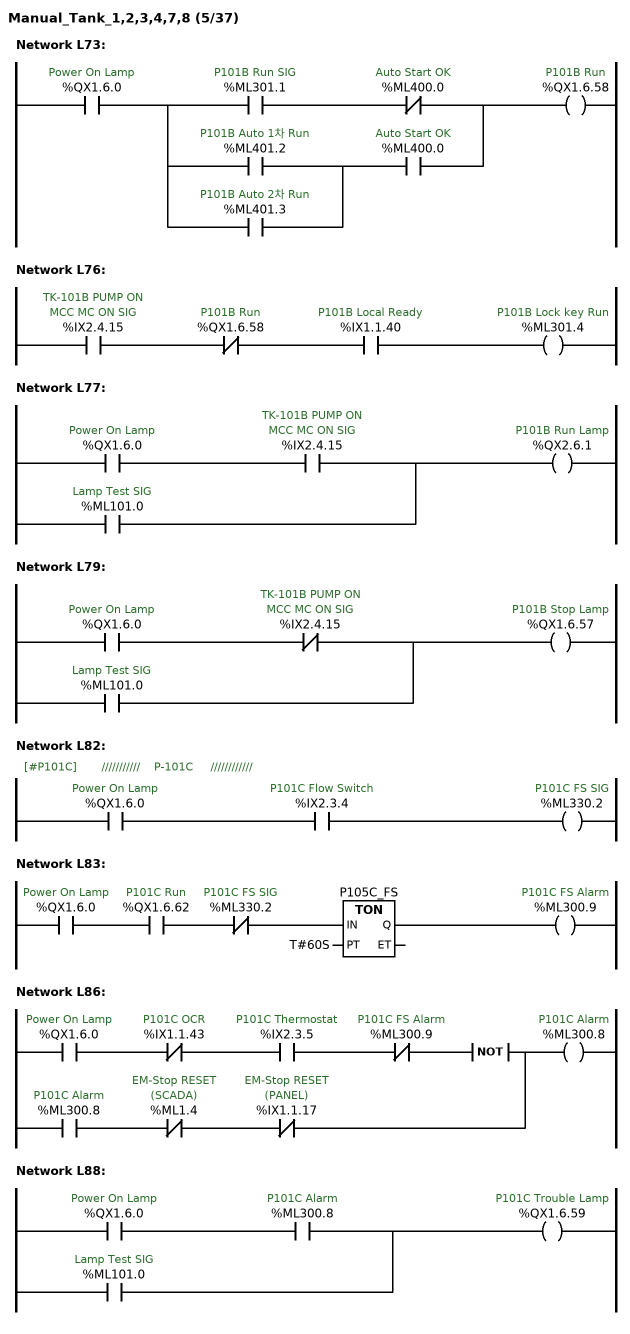
(* Rung L73 *)
%QX1.6.58 := %QX1.6.0 AND ((%ML301.1 AND NOT %ML400.0) OR ((%ML401.2 OR %ML401.3) AND %ML400.0));
(* Rung L76 *)
%ML301.4 := %IX2.4.15 AND NOT %QX1.6.58 AND %IX1.1.40;
(* Rung L77 *)
%QX2.6.1 := (%QX1.6.0 AND %IX2.4.15) OR %ML101.0;
(* Rung L79 *)
%QX1.6.57 := (%QX1.6.0 AND NOT %IX2.4.15) OR %ML101.0;
(* [#P101C]       ///////////    P-101C     //////////// *)
(* Rung L82 *)
%ML330.2 := %QX1.6.0 AND %IX2.3.4;
(* Rung L83 *)
P105C_FS(IN := %QX1.6.0 AND %QX1.6.62 AND NOT %ML330.2, PT := T#60S);
%ML300.9 := P105C_FS.Q;
(* Rung L86 *)
%ML300.8 := NOT (%QX1.6.0 AND NOT %IX1.1.43 AND %IX2.3.5 AND NOT %ML300.9) OR (%ML300.8 AND NOT %ML1.4 AND NOT %IX1.1.17);
(* Rung L88 *)
%QX1.6.59 := (%QX1.6.0 AND %ML300.8) OR %ML101.0;

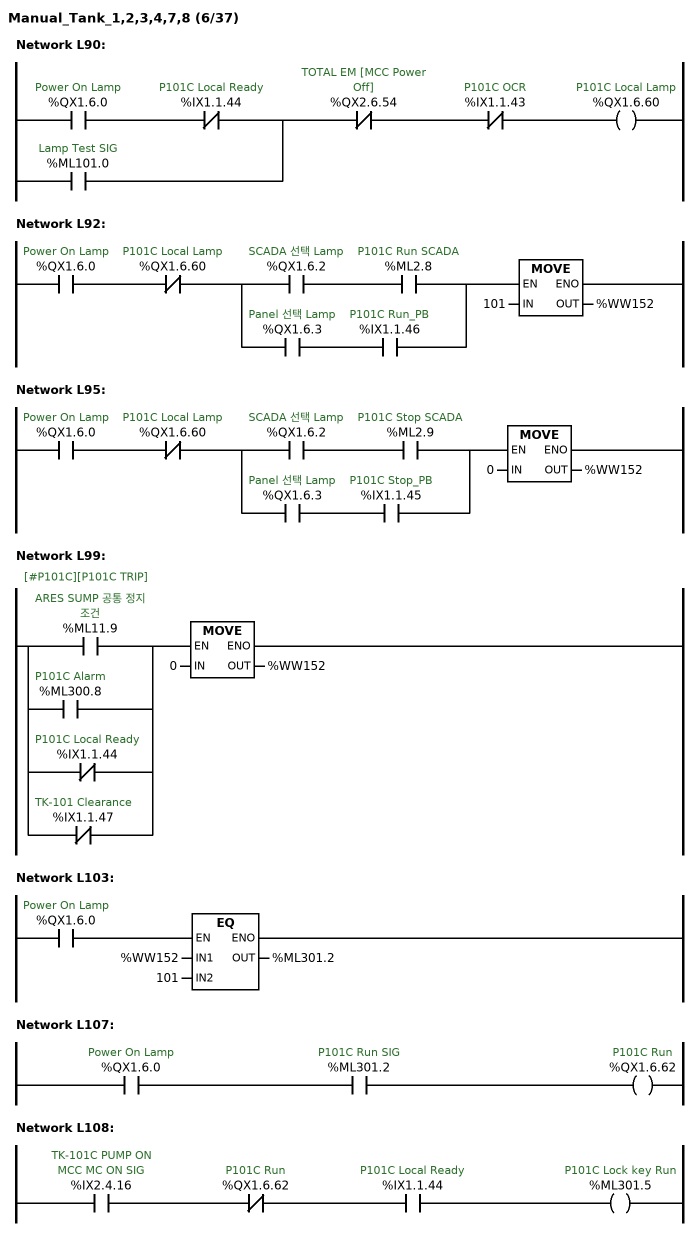
(* Rung L90 *)
%QX1.6.60 := ((%QX1.6.0 AND NOT %IX1.1.44) OR %ML101.0) AND NOT %QX2.6.54 AND NOT %IX1.1.43;
(* Rung L92 *)
IF %QX1.6.0 AND NOT %QX1.6.60 AND ((%QX1.6.2 AND %ML2.8) OR (%QX1.6.3 AND %IX1.1.46)) THEN
    %WW152 := 101;
END_IF;
(* Rung L95 *)
IF %QX1.6.0 AND NOT %QX1.6.60 AND ((%QX1.6.2 AND %ML2.9) OR (%QX1.6.3 AND %IX1.1.45)) THEN
    %WW152 := 0;
END_IF;
(* [#P101C][P101C TRIP] *)
(* Rung L99 *)
IF %ML11.9 OR %ML300.8 OR NOT %IX1.1.44 OR NOT %IX1.1.47 THEN %WW152 := 0; END_IF;
(* Rung L103 *)
IF %QX1.6.0 THEN %ML301.2 := %WW152 = 101; END_IF;
(* Rung L107 *)
%QX1.6.62 := %QX1.6.0 AND %ML301.2;
(* Rung L108 *)
%ML301.5 := %IX2.4.16 AND NOT %QX1.6.62 AND %IX1.1.44;

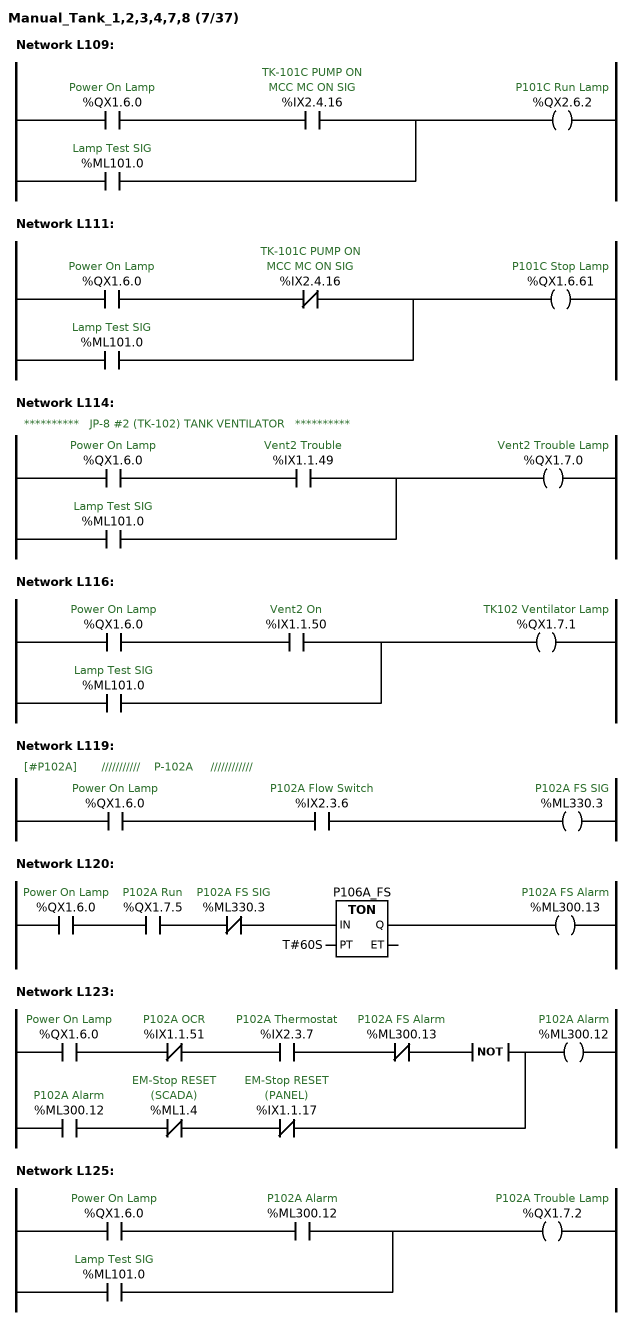
(* Rung L109 *)
%QX2.6.2 := (%QX1.6.0 AND %IX2.4.16) OR %ML101.0;
(* Rung L111 *)
%QX1.6.61 := (%QX1.6.0 AND NOT %IX2.4.16) OR %ML101.0;
(* **********   JP-8 #2 (TK-102) TANK VENTILATOR   ********** *)
(* Rung L114 *)
%QX1.7.0 := (%QX1.6.0 AND %IX1.1.49) OR %ML101.0;
(* Rung L116 *)
%QX1.7.1 := (%QX1.6.0 AND %IX1.1.50) OR %ML101.0;
(* [#P102A]       ///////////    P-102A     //////////// *)
(* Rung L119 *)
%ML330.3 := %QX1.6.0 AND %IX2.3.6;
(* Rung L120 *)
P106A_FS(IN := %QX1.6.0 AND %QX1.7.5 AND NOT %ML330.3, PT := T#60S);
%ML300.13 := P106A_FS.Q;
(* Rung L123 *)
%ML300.12 := NOT (%QX1.6.0 AND NOT %IX1.1.51 AND %IX2.3.7 AND NOT %ML300.13) OR (%ML300.12 AND NOT %ML1.4 AND NOT %IX1.1.17);
(* Rung L125 *)
%QX1.7.2 := (%QX1.6.0 AND %ML300.12) OR %ML101.0;

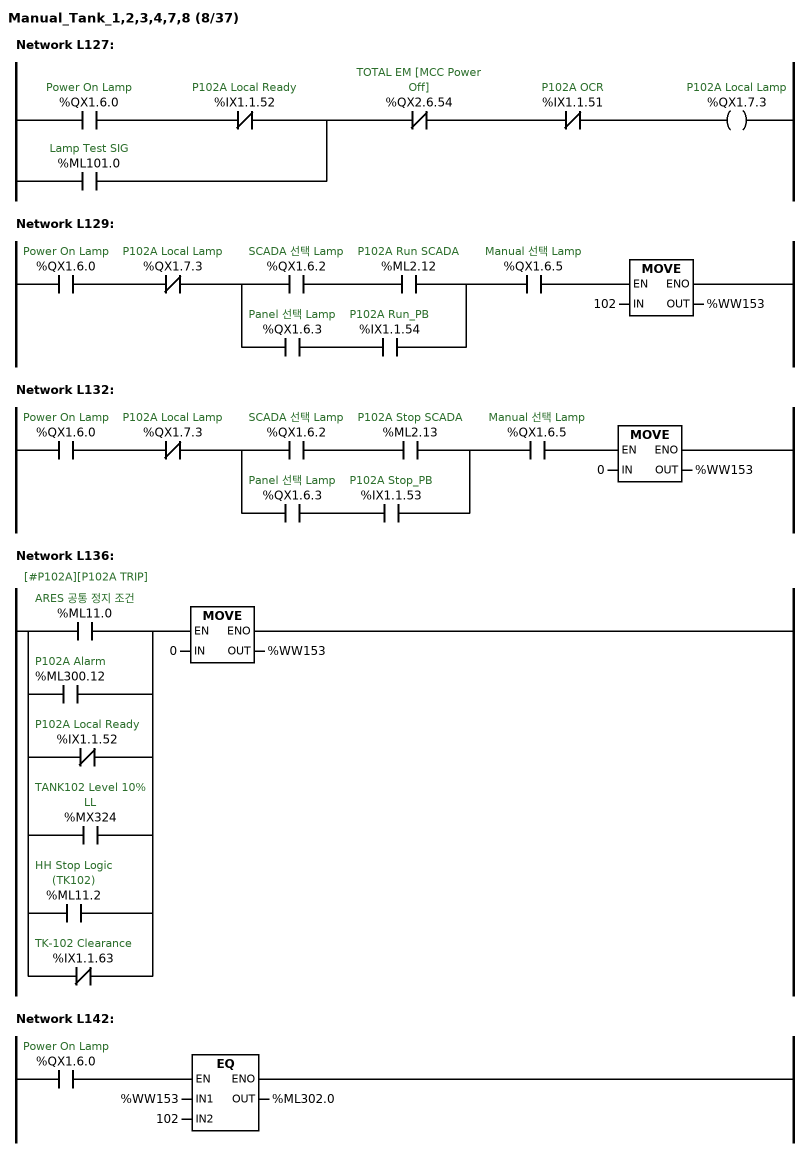
(* Rung L127 *)
%QX1.7.3 := ((%QX1.6.0 AND NOT %IX1.1.52) OR %ML101.0) AND NOT %QX2.6.54 AND NOT %IX1.1.51;
(* Rung L129 *)
IF %QX1.6.0 AND NOT %QX1.7.3 AND ((%QX1.6.2 AND %ML2.12) OR (%QX1.6.3 AND %IX1.1.54)) AND %QX1.6.5 THEN
    %WW153 := 102;
END_IF;
(* Rung L132 *)
IF %QX1.6.0 AND NOT %QX1.7.3 AND ((%QX1.6.2 AND %ML2.13) OR (%QX1.6.3 AND %IX1.1.53)) AND %QX1.6.5 THEN
    %WW153 := 0;
END_IF;
(* [#P102A][P102A TRIP] *)
(* Rung L136 *)
IF %ML11.0 OR %ML300.12 OR NOT %IX1.1.52 OR %MX324 OR %ML11.2 OR NOT %IX1.1.63 THEN %WW153 := 0; END_IF;
(* Rung L142 *)
IF %QX1.6.0 THEN %ML302.0 := %WW153 = 102; END_IF;

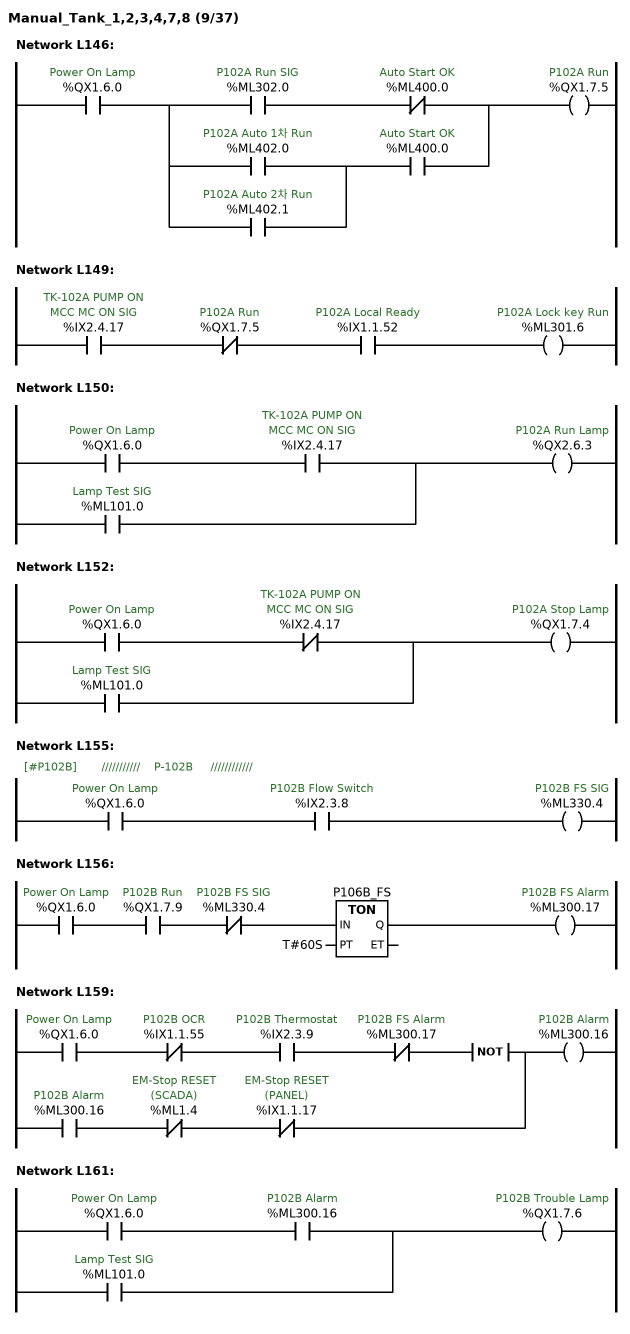
(* Rung L146 *)
%QX1.7.5 := %QX1.6.0 AND ((%ML302.0 AND NOT %ML400.0) OR ((%ML402.0 OR %ML402.1) AND %ML400.0));
(* Rung L149 *)
%ML301.6 := %IX2.4.17 AND NOT %QX1.7.5 AND %IX1.1.52;
(* Rung L150 *)
%QX2.6.3 := (%QX1.6.0 AND %IX2.4.17) OR %ML101.0;
(* Rung L152 *)
%QX1.7.4 := (%QX1.6.0 AND NOT %IX2.4.17) OR %ML101.0;
(* [#P102B]       ///////////    P-102B     //////////// *)
(* Rung L155 *)
%ML330.4 := %QX1.6.0 AND %IX2.3.8;
(* Rung L156 *)
P106B_FS(IN := %QX1.6.0 AND %QX1.7.9 AND NOT %ML330.4, PT := T#60S);
%ML300.17 := P106B_FS.Q;
(* Rung L159 *)
%ML300.16 := NOT (%QX1.6.0 AND NOT %IX1.1.55 AND %IX2.3.9 AND NOT %ML300.17) OR (%ML300.16 AND NOT %ML1.4 AND NOT %IX1.1.17);
(* Rung L161 *)
%QX1.7.6 := (%QX1.6.0 AND %ML300.16) OR %ML101.0;

